SPLINE
SPL {X  -134.737, Y  +296.229, Z    +0.000, E1  +312.110, E3 -135435.927}
SPL {X  -154.917, Y  +342.531, Z    +0.000, E1  +328.797, E3 -135454.495}
SPL {X  -159.440, Y  +369.246, Z    +0.000, E1  +346.542, E3 -135458.394}
SPL {X  -159.987, Y  +381.470, Z    +0.000, E1  +357.024, E3 -135458.993}
SPL {X  -159.990, Y  +384.500, Z    +0.000, E1  +360.000, E3 -135459.026}
SPL {X  -159.990, Y  +386.323, Z    +0.000, E1  +363.079, E3 -135459.048}
SPL {X  -159.990, Y  +390.285, Z    +0.000, E1  +371.315, E3 -135459.169}
SPL {X  -159.990, Y  +394.559, Z    +0.000, E1  +380.770, E3 -135459.431}
SPL {X  -159.990, Y  +399.334, Z    +0.000, E1  +390.876, E3 -135459.870}
SPL {X  -159.990, Y  +405.006, Z    +0.000, E1  +400.810, E3 -135460.588}
SPL {X  -159.990, Y  +415.193, Z    +0.000, E1  +412.724, E3 -135462.475}
SPL {X  -159.990, Y  +465.395, Z    +0.000, E1  +428.959, E3 -135477.563}
SPL {X  -159.990, Y  +657.157, Z    +0.000, E1  +432.499, E3 -135573.960}
SPL {X  -159.693, Y  +681.249, Z    +0.000, E1  +432.488, E3 -135590.354}
SPL {X  -157.599, Y  +699.059, Z    +0.000, E1  +432.249, E3 -135604.514}
SPL {X  -155.217, Y  +710.289, Z    +0.000, E1  +431.989, E3 -135614.530}
SPL {X  -152.611, Y  +719.527, Z    +0.000, E1  +431.702, E3 -135623.352}
SPL {X  -149.536, Y  +728.383, Z    +0.000, E1  +431.359, E3 -135632.331}
SPL {X  -146.250, Y  +736.367, Z    +0.000, E1  +430.965, E3 -135640.885}
SPL {X  -143.481, Y  +742.281, Z    +0.000, E1  +430.623, E3 -135647.480}
SPL {X  -140.071, Y  +748.811, Z    +0.000, E1  +430.193, E3 -135654.992}
SPL {X  -136.578, Y  +754.826, Z    +0.000, E1  +429.723, E3 -135662.122}
SPL {X  -132.176, Y  +761.646, Z    +0.000, E1  +429.128, E3 -135670.365}
SPL {X  -127.941, Y  +767.561, Z    +0.000, E1  +428.475, E3 -135677.673}
SPL {X  -124.983, Y  +771.380, Z    +0.000, E1  +428.003, E3 -135682.392}
SPL {X  -122.624, Y  +774.263, Z    +0.000, E1  +427.622, E3 -135685.915}
SPL {X   -84.435, Y  +807.395, Z    +0.000, E1  +415.948, E3 -135796.919}
ENDSPLINE

SPLINE
SPL {X  -119.703, Y  +777.650, Z    +0.000, E1  +411.831, E3 -135960.926}
SPL {X  -145.184, Y  +738.720, Z    +0.000, E1  +403.488, E3 -135987.484}
SPL {X  -156.175, Y  +706.232, Z    +0.000, E1  +388.819, E3 -135996.369}
SPL {X  -159.337, Y  +685.942, Z    +0.000, E1  +374.672, E3 -135998.920}
SPL {X  -159.962, Y  +674.468, Z    +0.000, E1  +364.846, E3 -135999.539}
SPL {X  -159.990, Y  +669.479, Z    +0.000, E1  +359.996, E3 -135999.613}
SPL {X  -159.990, Y  +667.035, Z    +0.000, E1  +355.461, E3 -135999.644}
SPL {X  -159.990, Y  +662.914, Z    +0.000, E1  +346.506, E3 -135999.782}
SPL {X  -159.990, Y  +658.254, Z    +0.000, E1  +335.847, E3 -136000.060}
SPL {X  -159.990, Y  +650.381, Z    +0.000, E1  +320.607, E3 -136000.912}
SPL {X  -159.990, Y  +638.701, Z    +0.000, E1  +306.047, E3 -136002.798}
SPL {X  -159.990, Y  +618.566, Z    +0.000, E1  +295.881, E3 -136008.306}
SPL {X  -159.990, Y  +582.261, Z    +0.000, E1  +290.657, E3 -136021.792}
SPL {X  -159.990, Y  +406.555, Z    +0.000, E1  +288.365, E3 -136118.038}
SPL {X  -159.990, Y  +385.723, Z    +0.000, E1  +288.390, E3 -136132.777}
SPL {X  -159.404, Y  +368.814, Z    +0.000, E1  +288.444, E3 -136145.306}
SPL {X  -157.440, Y  +354.048, Z    +0.000, E1  +288.658, E3 -136157.779}
SPL {X  -155.889, Y  +346.508, Z    +0.000, E1  +289.539, E3 -136171.327}
SPL {X  -154.332, Y  +340.328, Z    +0.000, E1  +289.976, E3 -136179.555}
SPL {X  -150.579, Y  +328.438, Z    +0.000, E1  +289.626, E3 -136185.274}
SPL {X  -146.933, Y  +319.195, Z    +0.000, E1  +289.770, E3 -136192.965}
SPL {X  -143.573, Y  +311.906, Z    +0.000, E1  +290.194, E3 -136201.275}
SPL {X  -139.693, Y  +304.508, Z    +0.000, E1  +290.699, E3 -136210.003}
SPL {X  -135.622, Y  +297.627, Z    +0.000, E1  +291.269, E3 -136218.411}
SPL {X  -131.165, Y  +290.889, Z    +0.000, E1  +291.906, E3 -136226.797}
SPL {X  -126.457, Y  +284.492, Z    +0.000, E1  +292.648, E3 -136234.882}
SPL {X  -123.432, Y  +280.710, Z    +0.000, E1  +293.170, E3 -136239.668}
SPL {X   -85.607, Y  +247.340, Z    +0.000, E1  +306.083, E3 -136381.389}
ENDSPLINE

SPLINE
SPL {X  -134.737, Y  +296.229, Z    +0.000, E1  +312.110, E3 -136524.162}
SPL {X  -154.917, Y  +342.531, Z    +0.000, E1  +328.797, E3 -136542.730}
SPL {X  -159.440, Y  +369.246, Z    +0.000, E1  +346.542, E3 -136546.629}
SPL {X  -159.987, Y  +381.470, Z    +0.000, E1  +357.024, E3 -136547.228}
SPL {X  -159.990, Y  +384.500, Z    +0.000, E1  +360.000, E3 -136547.261}
SPL {X  -159.990, Y  +386.323, Z    +0.000, E1  +363.079, E3 -136547.283}
SPL {X  -159.990, Y  +390.285, Z    +0.000, E1  +371.315, E3 -136547.404}
SPL {X  -159.990, Y  +394.559, Z    +0.000, E1  +380.770, E3 -136547.666}
SPL {X  -159.990, Y  +402.118, Z    +0.000, E1  +395.793, E3 -136548.457}
SPL {X  -159.990, Y  +415.193, Z    +0.000, E1  +412.724, E3 -136550.710}
SPL {X  -159.990, Y  +465.395, Z    +0.000, E1  +428.959, E3 -136565.799}
SPL {X  -159.990, Y  +652.170, Z    +0.000, E1  +432.485, E3 -136658.894}
SPL {X  -159.990, Y  +670.864, Z    +0.000, E1  +432.509, E3 -136671.342}
SPL {X  -159.251, Y  +686.856, Z    +0.000, E1  +432.412, E3 -136682.884}
SPL {X  -157.599, Y  +699.059, Z    +0.000, E1  +432.249, E3 -136692.749}
SPL {X  -155.217, Y  +710.289, Z    +0.000, E1  +431.989, E3 -136702.766}
SPL {X  -152.611, Y  +719.527, Z    +0.000, E1  +431.702, E3 -136711.587}
SPL {X  -149.536, Y  +728.383, Z    +0.000, E1  +431.359, E3 -136720.566}
SPL {X  -146.250, Y  +736.367, Z    +0.000, E1  +430.965, E3 -136729.120}
SPL {X  -143.481, Y  +742.281, Z    +0.000, E1  +430.623, E3 -136735.716}
SPL {X  -140.071, Y  +748.811, Z    +0.000, E1  +430.193, E3 -136743.227}
SPL {X  -136.578, Y  +754.826, Z    +0.000, E1  +429.723, E3 -136750.357}
SPL {X  -133.265, Y  +760.028, Z    +0.000, E1  +429.258, E3 -136756.658}
SPL {X  -129.890, Y  +764.909, Z    +0.000, E1  +428.775, E3 -136762.628}
SPL {X  -125.802, Y  +770.346, Z    +0.000, E1  +428.156, E3 -136769.328}
SPL {X  -122.624, Y  +774.263, Z    +0.000, E1  +427.622, E3 -136774.150}
SPL {X   -84.435, Y  +807.395, Z    +0.000, E1  +415.948, E3 -136885.155}
ENDSPLINE

SPLINE
SPL {X  -119.703, Y  +777.650, Z    +0.000, E1  +411.831, E3 -137049.161}
SPL {X  -145.184, Y  +738.720, Z    +0.000, E1  +403.488, E3 -137075.719}
SPL {X  -156.175, Y  +706.232, Z    +0.000, E1  +388.819, E3 -137084.604}
SPL {X  -159.337, Y  +685.942, Z    +0.000, E1  +374.672, E3 -137087.155}
SPL {X  -159.962, Y  +674.468, Z    +0.000, E1  +364.846, E3 -137087.774}
SPL {X  -159.990, Y  +669.479, Z    +0.000, E1  +359.996, E3 -137087.848}
SPL {X  -159.990, Y  +667.035, Z    +0.000, E1  +355.461, E3 -137087.879}
SPL {X  -159.990, Y  +662.914, Z    +0.000, E1  +346.506, E3 -137088.018}
SPL {X  -159.990, Y  +658.254, Z    +0.000, E1  +335.847, E3 -137088.295}
SPL {X  -159.990, Y  +652.944, Z    +0.000, E1  +324.878, E3 -137088.799}
SPL {X  -159.990, Y  +642.509, Z    +0.000, E1  +309.910, E3 -137090.371}
SPL {X  -159.990, Y  +618.566, Z    +0.000, E1  +295.881, E3 -137096.541}
SPL {X  -159.990, Y  +584.545, Z    +0.000, E1  +290.812, E3 -137109.076}
SPL {X  -159.990, Y  +578.002, Z    +0.000, E1  +290.393, E3 -137111.800}
SPL {X  -159.990, Y  +426.570, Z    +0.000, E1  +288.401, E3 -137192.290}
SPL {X  -159.990, Y  +405.946, Z    +0.000, E1  +288.370, E3 -137206.720}
SPL {X  -159.967, Y  +379.776, Z    +0.000, E1  +288.366, E3 -137225.167}
SPL {X  -158.535, Y  +360.970, Z    +0.000, E1  +288.540, E3 -137239.989}
SPL {X  -156.277, Y  +348.230, Z    +0.000, E1  +288.789, E3 -137251.332}
SPL {X  -155.351, Y  +344.251, Z    +0.000, E1  +289.996, E3 -137265.124}
SPL {X  -150.579, Y  +328.438, Z    +0.000, E1  +289.626, E3 -137273.509}
SPL {X  -146.933, Y  +319.195, Z    +0.000, E1  +289.770, E3 -137281.200}
SPL {X  -143.573, Y  +311.906, Z    +0.000, E1  +290.194, E3 -137289.510}
SPL {X  -139.693, Y  +304.508, Z    +0.000, E1  +290.699, E3 -137298.239}
SPL {X  -135.622, Y  +297.627, Z    +0.000, E1  +291.269, E3 -137306.647}
SPL {X  -131.165, Y  +290.889, Z    +0.000, E1  +291.906, E3 -137315.032}
SPL {X  -126.457, Y  +284.492, Z    +0.000, E1  +292.648, E3 -137323.118}
SPL {X  -123.432, Y  +280.710, Z    +0.000, E1  +293.170, E3 -137327.903}
SPL {X   -85.607, Y  +247.340, Z    +0.000, E1  +306.083, E3 -137469.625}
ENDSPLINE

SPLINE
SPL {X  -134.737, Y  +296.229, Z    +0.000, E1  +312.110, E3 -137612.398}
SPL {X  -154.917, Y  +342.531, Z    +0.000, E1  +328.797, E3 -137630.965}
SPL {X  -159.440, Y  +369.246, Z    +0.000, E1  +346.542, E3 -137634.864}
SPL {X  -159.957, Y  +379.264, Z    +0.000, E1  +355.091, E3 -137635.421}
SPL {X  -159.990, Y  +384.670, Z    +0.000, E1  +360.079, E3 -137635.498}
SPL {X  -159.990, Y  +389.248, Z    +0.000, E1  +368.879, E3 -137635.602}
SPL {X  -159.990, Y  +394.559, Z    +0.000, E1  +380.770, E3 -137635.901}
SPL {X  -159.990, Y  +402.118, Z    +0.000, E1  +395.793, E3 -137636.693}
SPL {X  -159.990, Y  +415.193, Z    +0.000, E1  +412.724, E3 -137638.945}
SPL {X  -159.990, Y  +465.395, Z    +0.000, E1  +428.959, E3 -137654.034}
SPL {X  -159.990, Y  +657.157, Z    +0.000, E1  +432.499, E3 -137750.431}
SPL {X  -159.947, Y  +675.227, Z    +0.000, E1  +432.487, E3 -137762.591}
SPL {X  -159.251, Y  +686.856, Z    +0.000, E1  +432.412, E3 -137771.119}
SPL {X  -157.599, Y  +699.059, Z    +0.000, E1  +432.249, E3 -137780.984}
SPL {X  -155.217, Y  +710.289, Z    +0.000, E1  +431.989, E3 -137791.001}
SPL {X  -152.611, Y  +719.527, Z    +0.000, E1  +431.702, E3 -137799.822}
SPL {X  -149.536, Y  +728.383, Z    +0.000, E1  +431.359, E3 -137808.801}
SPL {X  -146.250, Y  +736.367, Z    +0.000, E1  +430.965, E3 -137817.356}
SPL {X  -143.481, Y  +742.281, Z    +0.000, E1  +430.623, E3 -137823.951}
SPL {X  -140.071, Y  +748.811, Z    +0.000, E1  +430.193, E3 -137831.463}
SPL {X  -136.578, Y  +754.826, Z    +0.000, E1  +429.723, E3 -137838.592}
SPL {X  -133.265, Y  +760.028, Z    +0.000, E1  +429.258, E3 -137844.893}
SPL {X  -129.890, Y  +764.909, Z    +0.000, E1  +428.775, E3 -137850.864}
SPL {X  -125.802, Y  +770.346, Z    +0.000, E1  +428.156, E3 -137857.563}
SPL {X  -122.624, Y  +774.263, Z    +0.000, E1  +427.622, E3 -137862.386}
SPL {X   -84.435, Y  +807.395, Z    +0.000, E1  +415.948, E3 -137973.390}
ENDSPLINE

SPLINE
SPL {X  -119.703, Y  +777.650, Z    +0.000, E1  +411.831, E3 -138137.397}
SPL {X  -145.184, Y  +738.720, Z    +0.000, E1  +403.488, E3 -138163.955}
SPL {X  -154.467, Y  +713.173, Z    +0.000, E1  +392.658, E3 -138171.550}
SPL {X  -157.530, Y  +699.446, Z    +0.000, E1  +384.482, E3 -138173.966}
SPL {X  -159.337, Y  +685.942, Z    +0.000, E1  +374.672, E3 -138175.391}
SPL {X  -159.962, Y  +674.468, Z    +0.000, E1  +364.846, E3 -138176.009}
SPL {X  -159.990, Y  +669.479, Z    +0.000, E1  +359.996, E3 -138176.083}
SPL {X  -159.990, Y  +667.035, Z    +0.000, E1  +355.461, E3 -138176.114}
SPL {X  -159.990, Y  +662.914, Z    +0.000, E1  +346.506, E3 -138176.253}
SPL {X  -159.990, Y  +658.254, Z    +0.000, E1  +335.847, E3 -138176.531}
SPL {X  -159.990, Y  +652.944, Z    +0.000, E1  +324.878, E3 -138177.034}
SPL {X  -159.990, Y  +642.509, Z    +0.000, E1  +309.910, E3 -138178.606}
SPL {X  -159.990, Y  +618.566, Z    +0.000, E1  +295.881, E3 -138184.777}
SPL {X  -159.990, Y  +582.261, Z    +0.000, E1  +290.657, E3 -138198.262}
SPL {X  -159.990, Y  +406.555, Z    +0.000, E1  +288.365, E3 -138294.509}
SPL {X  -159.990, Y  +385.723, Z    +0.000, E1  +288.390, E3 -138309.247}
SPL {X  -159.700, Y  +372.863, Z    +0.000, E1  +288.430, E3 -138318.653}
SPL {X  -158.535, Y  +360.970, Z    +0.000, E1  +288.540, E3 -138328.224}
SPL {X  -156.277, Y  +348.230, Z    +0.000, E1  +288.789, E3 -138339.567}
SPL {X  -155.351, Y  +344.251, Z    +0.000, E1  +289.996, E3 -138353.359}
SPL {X  -150.579, Y  +328.438, Z    +0.000, E1  +289.626, E3 -138361.744}
SPL {X  -146.933, Y  +319.195, Z    +0.000, E1  +289.770, E3 -138369.435}
SPL {X  -143.573, Y  +311.906, Z    +0.000, E1  +290.194, E3 -138377.746}
SPL {X  -140.547, Y  +306.057, Z    +0.000, E1  +290.601, E3 -138384.638}
SPL {X  -137.438, Y  +300.600, Z    +0.000, E1  +291.016, E3 -138391.232}
SPL {X  -133.397, Y  +294.172, Z    +0.000, E1  +291.584, E3 -138399.167}
SPL {X  -128.822, Y  +287.623, Z    +0.000, E1  +292.271, E3 -138407.391}
SPL {X  -124.502, Y  +282.021, Z    +0.000, E1  +292.965, E3 -138414.465}
SPL {X   -85.607, Y  +247.340, Z    +0.000, E1  +306.083, E3 -138557.860}
ENDSPLINE

SPLINE
SPL {X  -119.557, Y  +276.184, Z    +0.000, E1  +308.968, E3 -138681.397}
SPL {X  -138.294, Y  +302.054, Z    +0.000, E1  +313.424, E3 -138704.719}
SPL {X  -153.211, Y  +336.421, Z    +0.000, E1  +325.738, E3 -138717.841}
SPL {X  -158.240, Y  +358.900, Z    +0.000, E1  +338.911, E3 -138722.046}
SPL {X  -159.674, Y  +372.451, Z    +0.000, E1  +349.222, E3 -138723.342}
SPL {X  -159.987, Y  +381.470, Z    +0.000, E1  +357.024, E3 -138723.699}
SPL {X  -159.990, Y  +384.761, Z    +0.000, E1  +360.257, E3 -138723.734}
SPL {X  -159.990, Y  +389.248, Z    +0.000, E1  +368.879, E3 -138723.838}
SPL {X  -159.990, Y  +394.559, Z    +0.000, E1  +380.770, E3 -138724.137}
SPL {X  -159.990, Y  +402.118, Z    +0.000, E1  +395.793, E3 -138724.928}
SPL {X  -159.990, Y  +415.193, Z    +0.000, E1  +412.724, E3 -138727.181}
SPL {X  -159.990, Y  +465.395, Z    +0.000, E1  +428.959, E3 -138742.269}
SPL {X  -159.990, Y  +657.157, Z    +0.000, E1  +432.499, E3 -138838.666}
SPL {X  -159.693, Y  +681.249, Z    +0.000, E1  +432.488, E3 -138855.060}
SPL {X  -157.599, Y  +699.059, Z    +0.000, E1  +432.249, E3 -138869.220}
SPL {X  -155.217, Y  +710.289, Z    +0.000, E1  +431.989, E3 -138879.236}
SPL {X  -152.611, Y  +719.527, Z    +0.000, E1  +431.702, E3 -138888.058}
SPL {X  -149.536, Y  +728.383, Z    +0.000, E1  +431.359, E3 -138897.037}
SPL {X  -146.250, Y  +736.367, Z    +0.000, E1  +430.965, E3 -138905.591}
SPL {X  -143.481, Y  +742.281, Z    +0.000, E1  +430.623, E3 -138912.186}
SPL {X  -140.071, Y  +748.811, Z    +0.000, E1  +430.193, E3 -138919.698}
SPL {X  -136.578, Y  +754.826, Z    +0.000, E1  +429.723, E3 -138926.827}
SPL {X  -133.265, Y  +760.028, Z    +0.000, E1  +429.258, E3 -138933.128}
SPL {X  -129.890, Y  +764.909, Z    +0.000, E1  +428.775, E3 -138939.099}
SPL {X  -125.802, Y  +770.346, Z    +0.000, E1  +428.156, E3 -138945.798}
SPL {X  -122.624, Y  +774.263, Z    +0.000, E1  +427.622, E3 -138950.621}
SPL {X   -84.435, Y  +807.395, Z    +0.000, E1  +415.948, E3 -139061.625}
ENDSPLINE

SPLINE
SPL {X  -119.703, Y  +777.650, Z    +0.000, E1  +411.831, E3 -139225.632}
SPL {X  -145.184, Y  +738.720, Z    +0.000, E1  +403.488, E3 -139252.190}
SPL {X  -156.175, Y  +706.232, Z    +0.000, E1  +388.819, E3 -139261.075}
SPL {X  -159.337, Y  +685.942, Z    +0.000, E1  +374.672, E3 -139263.626}
SPL {X  -159.900, Y  +676.871, Z    +0.000, E1  +366.955, E3 -139264.174}
SPL {X  -159.990, Y  +669.634, Z    +0.000, E1  +360.285, E3 -139264.318}
SPL {X  -159.990, Y  +667.035, Z    +0.000, E1  +355.461, E3 -139264.349}
SPL {X  -159.990, Y  +662.914, Z    +0.000, E1  +346.506, E3 -139264.488}
SPL {X  -159.990, Y  +658.254, Z    +0.000, E1  +335.847, E3 -139264.766}
SPL {X  -159.990, Y  +652.944, Z    +0.000, E1  +324.878, E3 -139265.270}
SPL {X  -159.990, Y  +642.509, Z    +0.000, E1  +309.910, E3 -139266.841}
SPL {X  -159.990, Y  +618.566, Z    +0.000, E1  +295.881, E3 -139273.012}
SPL {X  -159.990, Y  +584.545, Z    +0.000, E1  +290.812, E3 -139285.547}
SPL {X  -159.990, Y  +578.002, Z    +0.000, E1  +290.393, E3 -139288.271}
SPL {X  -159.990, Y  +426.570, Z    +0.000, E1  +288.401, E3 -139368.761}
SPL {X  -159.990, Y  +405.946, Z    +0.000, E1  +288.370, E3 -139383.191}
SPL {X  -159.967, Y  +379.776, Z    +0.000, E1  +288.366, E3 -139401.637}
SPL {X  -158.535, Y  +360.970, Z    +0.000, E1  +288.540, E3 -139416.459}
SPL {X  -156.882, Y  +351.118, Z    +0.000, E1  +288.737, E3 -139425.171}
SPL {X  -155.538, Y  +345.018, Z    +0.000, E1  +288.891, E3 -139430.878}
SPL {X  -155.351, Y  +344.251, Z    +0.000, E1  +289.996, E3 -139441.594}
SPL {X  -150.579, Y  +328.438, Z    +0.000, E1  +289.626, E3 -139449.980}
SPL {X  -146.933, Y  +319.195, Z    +0.000, E1  +289.770, E3 -139457.671}
SPL {X  -143.573, Y  +311.906, Z    +0.000, E1  +290.194, E3 -139465.981}
SPL {X  -140.547, Y  +306.057, Z    +0.000, E1  +290.601, E3 -139472.873}
SPL {X  -137.438, Y  +300.600, Z    +0.000, E1  +291.016, E3 -139479.467}
SPL {X  -133.397, Y  +294.172, Z    +0.000, E1  +291.584, E3 -139487.402}
SPL {X  -128.822, Y  +287.623, Z    +0.000, E1  +292.271, E3 -139495.627}
SPL {X  -124.502, Y  +282.021, Z    +0.000, E1  +292.965, E3 -139502.701}
SPL {X   -85.607, Y  +247.340, Z    +0.000, E1  +306.083, E3 -139646.095}
ENDSPLINE

SPLINE
SPL {X  -134.737, Y  +296.229, Z    +0.000, E1  +312.110, E3 -139788.868}
SPL {X  -153.211, Y  +336.421, Z    +0.000, E1  +325.738, E3 -139806.076}
SPL {X  -158.240, Y  +358.900, Z    +0.000, E1  +338.911, E3 -139810.281}
SPL {X  -159.854, Y  +375.896, Z    +0.000, E1  +352.019, E3 -139811.747}
SPL {X  -159.990, Y  +384.398, Z    +0.000, E1  +359.828, E3 -139811.967}
SPL {X  -159.990, Y  +386.323, Z    +0.000, E1  +363.079, E3 -139811.989}
SPL {X  -159.990, Y  +390.285, Z    +0.000, E1  +371.315, E3 -139812.110}
SPL {X  -159.990, Y  +394.559, Z    +0.000, E1  +380.770, E3 -139812.372}
SPL {X  -159.990, Y  +399.334, Z    +0.000, E1  +390.876, E3 -139812.811}
SPL {X  -159.990, Y  +405.006, Z    +0.000, E1  +400.810, E3 -139813.529}
SPL {X  -159.990, Y  +415.193, Z    +0.000, E1  +412.724, E3 -139815.416}
SPL {X  -159.990, Y  +465.395, Z    +0.000, E1  +428.959, E3 -139830.505}
SPL {X  -159.990, Y  +657.157, Z    +0.000, E1  +432.499, E3 -139926.901}
SPL {X  -159.693, Y  +681.249, Z    +0.000, E1  +432.488, E3 -139943.295}
SPL {X  -157.599, Y  +699.059, Z    +0.000, E1  +432.249, E3 -139957.455}
SPL {X  -155.217, Y  +710.289, Z    +0.000, E1  +431.989, E3 -139967.472}
SPL {X  -152.611, Y  +719.527, Z    +0.000, E1  +431.702, E3 -139976.293}
SPL {X  -149.536, Y  +728.383, Z    +0.000, E1  +431.359, E3 -139985.272}
SPL {X  -146.250, Y  +736.367, Z    +0.000, E1  +430.965, E3 -139993.826}
SPL {X  -143.481, Y  +742.281, Z    +0.000, E1  +430.623, E3 -140000.422}
SPL {X  -140.071, Y  +748.811, Z    +0.000, E1  +430.193, E3 -140007.933}
SPL {X  -136.578, Y  +754.826, Z    +0.000, E1  +429.723, E3 -140015.063}
SPL {X  -133.265, Y  +760.028, Z    +0.000, E1  +429.258, E3 -140021.364}
SPL {X  -129.890, Y  +764.909, Z    +0.000, E1  +428.775, E3 -140027.334}
SPL {X  -125.802, Y  +770.346, Z    +0.000, E1  +428.156, E3 -140034.033}
SPL {X  -122.624, Y  +774.263, Z    +0.000, E1  +427.622, E3 -140038.856}
SPL {X   -84.435, Y  +807.395, Z    +0.000, E1  +415.948, E3 -140149.861}
ENDSPLINE

SPLINE
SPL {X  -119.703, Y  +777.650, Z    +0.000, E1  +411.831, E3 -140313.867}
SPL {X  -145.184, Y  +738.720, Z    +0.000, E1  +403.488, E3 -140340.425}
SPL {X  -156.175, Y  +706.232, Z    +0.000, E1  +388.819, E3 -140349.310}
SPL {X  -159.337, Y  +685.942, Z    +0.000, E1  +374.672, E3 -140351.861}
SPL {X  -159.900, Y  +676.871, Z    +0.000, E1  +366.955, E3 -140352.409}
SPL {X  -159.990, Y  +669.634, Z    +0.000, E1  +360.285, E3 -140352.553}
SPL {X  -159.990, Y  +667.035, Z    +0.000, E1  +355.461, E3 -140352.585}
SPL {X  -159.990, Y  +662.914, Z    +0.000, E1  +346.506, E3 -140352.724}
SPL {X  -159.990, Y  +658.254, Z    +0.000, E1  +335.847, E3 -140353.001}
SPL {X  -159.990, Y  +652.944, Z    +0.000, E1  +324.878, E3 -140353.505}
SPL {X  -159.990, Y  +646.557, Z    +0.000, E1  +314.610, E3 -140354.372}
SPL {X  -159.990, Y  +638.701, Z    +0.000, E1  +306.047, E3 -140355.739}
SPL {X  -159.990, Y  +618.566, Z    +0.000, E1  +295.881, E3 -140361.247}
SPL {X  -159.990, Y  +582.261, Z    +0.000, E1  +290.657, E3 -140374.733}
SPL {X  -159.990, Y  +414.423, Z    +0.000, E1  +288.398, E3 -140465.516}
SPL {X  -159.990, Y  +400.357, Z    +0.000, E1  +288.396, E3 -140475.427}
SPL {X  -159.990, Y  +385.723, Z    +0.000, E1  +288.390, E3 -140485.718}
SPL {X  -159.404, Y  +368.814, Z    +0.000, E1  +288.444, E3 -140498.247}
SPL {X  -157.440, Y  +354.048, Z    +0.000, E1  +288.658, E3 -140510.720}
SPL {X  -155.889, Y  +346.508, Z    +0.000, E1  +289.539, E3 -140524.268}
SPL {X  -154.332, Y  +340.328, Z    +0.000, E1  +289.976, E3 -140532.496}
SPL {X  -150.579, Y  +328.438, Z    +0.000, E1  +289.626, E3 -140538.215}
SPL {X  -146.933, Y  +319.195, Z    +0.000, E1  +289.770, E3 -140545.906}
SPL {X  -143.573, Y  +311.906, Z    +0.000, E1  +290.194, E3 -140554.216}
SPL {X  -139.693, Y  +304.508, Z    +0.000, E1  +290.699, E3 -140562.945}
SPL {X  -135.622, Y  +297.627, Z    +0.000, E1  +291.269, E3 -140571.353}
SPL {X  -132.531, Y  +292.877, Z    +0.000, E1  +291.734, E3 -140577.288}
SPL {X  -128.822, Y  +287.623, Z    +0.000, E1  +292.271, E3 -140583.862}
SPL {X  -124.502, Y  +282.021, Z    +0.000, E1  +292.965, E3 -140590.936}
SPL {X   -85.607, Y  +247.340, Z    +0.000, E1  +306.083, E3 -140734.331}
ENDSPLINE

SPLINE
SPL {X  -134.737, Y  +296.229, Z    +0.000, E1  +312.110, E3 -140877.103}
SPL {X  -154.917, Y  +342.531, Z    +0.000, E1  +328.797, E3 -140895.671}
SPL {X  -159.440, Y  +369.246, Z    +0.000, E1  +346.542, E3 -140899.570}
SPL {X  -159.987, Y  +381.470, Z    +0.000, E1  +357.024, E3 -140900.169}
SPL {X  -159.990, Y  +384.500, Z    +0.000, E1  +360.000, E3 -140900.203}
SPL {X  -159.990, Y  +386.323, Z    +0.000, E1  +363.079, E3 -140900.224}
SPL {X  -159.990, Y  +390.285, Z    +0.000, E1  +371.315, E3 -140900.345}
SPL {X  -159.990, Y  +394.559, Z    +0.000, E1  +380.770, E3 -140900.607}
SPL {X  -159.990, Y  +402.118, Z    +0.000, E1  +395.793, E3 -140901.399}
SPL {X  -159.990, Y  +415.193, Z    +0.000, E1  +412.724, E3 -140903.651}
SPL {X  -159.990, Y  +465.395, Z    +0.000, E1  +428.959, E3 -140918.740}
SPL {X  -159.990, Y  +657.157, Z    +0.000, E1  +432.499, E3 -141015.137}
SPL {X  -159.693, Y  +681.249, Z    +0.000, E1  +432.488, E3 -141031.531}
SPL {X  -157.599, Y  +699.059, Z    +0.000, E1  +432.249, E3 -141045.690}
SPL {X  -155.217, Y  +710.289, Z    +0.000, E1  +431.989, E3 -141055.707}
SPL {X  -152.611, Y  +719.527, Z    +0.000, E1  +431.702, E3 -141064.528}
SPL {X  -149.536, Y  +728.383, Z    +0.000, E1  +431.359, E3 -141073.507}
SPL {X  -146.250, Y  +736.367, Z    +0.000, E1  +430.965, E3 -141082.061}
SPL {X  -143.481, Y  +742.281, Z    +0.000, E1  +430.623, E3 -141088.657}
SPL {X  -140.071, Y  +748.811, Z    +0.000, E1  +430.193, E3 -141096.169}
SPL {X  -136.578, Y  +754.826, Z    +0.000, E1  +429.723, E3 -141103.298}
SPL {X  -133.265, Y  +760.028, Z    +0.000, E1  +429.258, E3 -141109.599}
SPL {X  -129.890, Y  +764.909, Z    +0.000, E1  +428.775, E3 -141115.570}
SPL {X  -125.802, Y  +770.346, Z    +0.000, E1  +428.156, E3 -141122.269}
SPL {X  -122.624, Y  +774.263, Z    +0.000, E1  +427.622, E3 -141127.091}
SPL {X   -84.435, Y  +807.395, Z    +0.000, E1  +415.948, E3 -141238.096}
ENDSPLINE

SPLINE
SPL {X  -119.703, Y  +777.650, Z    +0.000, E1  +411.831, E3 -141402.103}
SPL {X  -145.184, Y  +738.720, Z    +0.000, E1  +403.488, E3 -141428.661}
SPL {X  -156.175, Y  +706.232, Z    +0.000, E1  +388.819, E3 -141437.545}
SPL {X  -159.337, Y  +685.942, Z    +0.000, E1  +374.672, E3 -141440.097}
SPL {X  -159.962, Y  +674.468, Z    +0.000, E1  +364.846, E3 -141440.715}
SPL {X  -159.990, Y  +669.479, Z    +0.000, E1  +359.996, E3 -141440.789}
SPL {X  -159.990, Y  +667.035, Z    +0.000, E1  +355.461, E3 -141440.820}
SPL {X  -159.990, Y  +662.914, Z    +0.000, E1  +346.506, E3 -141440.959}
SPL {X  -159.990, Y  +658.254, Z    +0.000, E1  +335.847, E3 -141441.237}
SPL {X  -159.990, Y  +652.944, Z    +0.000, E1  +324.878, E3 -141441.740}
SPL {X  -159.990, Y  +642.509, Z    +0.000, E1  +309.910, E3 -141443.312}
SPL {X  -159.990, Y  +618.566, Z    +0.000, E1  +295.881, E3 -141449.482}
SPL {X  -159.990, Y  +584.545, Z    +0.000, E1  +290.812, E3 -141462.018}
SPL {X  -159.990, Y  +578.002, Z    +0.000, E1  +290.393, E3 -141464.741}
SPL {X  -159.990, Y  +426.570, Z    +0.000, E1  +288.401, E3 -141545.231}
SPL {X  -159.990, Y  +405.946, Z    +0.000, E1  +288.370, E3 -141559.661}
SPL {X  -159.967, Y  +379.776, Z    +0.000, E1  +288.366, E3 -141578.108}
SPL {X  -158.535, Y  +360.970, Z    +0.000, E1  +288.540, E3 -141592.930}
SPL {X  -156.277, Y  +348.230, Z    +0.000, E1  +288.789, E3 -141604.273}
SPL {X  -155.351, Y  +344.251, Z    +0.000, E1  +289.996, E3 -141618.065}
SPL {X  -150.579, Y  +328.438, Z    +0.000, E1  +289.626, E3 -141626.450}
SPL {X  -146.933, Y  +319.195, Z    +0.000, E1  +289.770, E3 -141634.141}
SPL {X  -143.573, Y  +311.906, Z    +0.000, E1  +290.194, E3 -141642.452}
SPL {X  -139.693, Y  +304.508, Z    +0.000, E1  +290.699, E3 -141651.180}
SPL {X  -135.622, Y  +297.627, Z    +0.000, E1  +291.269, E3 -141659.588}
SPL {X  -131.165, Y  +290.889, Z    +0.000, E1  +291.906, E3 -141667.973}
SPL {X  -126.457, Y  +284.492, Z    +0.000, E1  +292.648, E3 -141676.059}
SPL {X  -123.432, Y  +280.710, Z    +0.000, E1  +293.170, E3 -141680.845}
SPL {X   -85.607, Y  +247.340, Z    +0.000, E1  +306.083, E3 -141822.566}
ENDSPLINE

SPLINE
SPL {X  -134.737, Y  +296.229, Z    +0.000, E1  +312.110, E3 -141965.339}
SPL {X  -154.917, Y  +342.531, Z    +0.000, E1  +328.797, E3 -141983.906}
SPL {X  -159.440, Y  +369.246, Z    +0.000, E1  +346.542, E3 -141987.806}
SPL {X  -159.987, Y  +381.470, Z    +0.000, E1  +357.024, E3 -141988.405}
SPL {X  -159.990, Y  +384.500, Z    +0.000, E1  +360.000, E3 -141988.438}
SPL {X  -159.990, Y  +386.323, Z    +0.000, E1  +363.079, E3 -141988.459}
SPL {X  -159.990, Y  +390.285, Z    +0.000, E1  +371.315, E3 -141988.580}
SPL {X  -159.990, Y  +394.559, Z    +0.000, E1  +380.770, E3 -141988.843}
SPL {X  -159.990, Y  +402.118, Z    +0.000, E1  +395.793, E3 -141989.634}
SPL {X  -159.990, Y  +415.193, Z    +0.000, E1  +412.724, E3 -141991.886}
SPL {X  -159.990, Y  +465.395, Z    +0.000, E1  +428.959, E3 -142006.975}
SPL {X  -159.990, Y  +657.157, Z    +0.000, E1  +432.499, E3 -142103.372}
SPL {X  -159.693, Y  +681.249, Z    +0.000, E1  +432.488, E3 -142119.766}
SPL {X  -157.599, Y  +699.059, Z    +0.000, E1  +432.249, E3 -142133.926}
SPL {X  -155.217, Y  +710.289, Z    +0.000, E1  +431.989, E3 -142143.942}
SPL {X  -152.611, Y  +719.527, Z    +0.000, E1  +431.702, E3 -142152.763}
SPL {X  -149.536, Y  +728.383, Z    +0.000, E1  +431.359, E3 -142161.743}
SPL {X  -146.250, Y  +736.367, Z    +0.000, E1  +430.965, E3 -142170.297}
SPL {X  -143.481, Y  +742.281, Z    +0.000, E1  +430.623, E3 -142176.892}
SPL {X  -140.071, Y  +748.811, Z    +0.000, E1  +430.193, E3 -142184.404}
SPL {X  -136.578, Y  +754.826, Z    +0.000, E1  +429.723, E3 -142191.533}
SPL {X  -133.265, Y  +760.028, Z    +0.000, E1  +429.258, E3 -142197.834}
SPL {X  -129.890, Y  +764.909, Z    +0.000, E1  +428.775, E3 -142203.805}
SPL {X  -125.802, Y  +770.346, Z    +0.000, E1  +428.156, E3 -142210.504}
SPL {X  -122.624, Y  +774.263, Z    +0.000, E1  +427.622, E3 -142215.327}
SPL {X   -84.435, Y  +807.395, Z    +0.000, E1  +415.948, E3 -142326.331}
ENDSPLINE

SPLINE
SPL {X  -119.703, Y  +777.650, Z    +0.000, E1  +411.831, E3 -142490.338}
SPL {X  -145.184, Y  +738.720, Z    +0.000, E1  +403.488, E3 -142516.896}
SPL {X  -156.175, Y  +706.232, Z    +0.000, E1  +388.819, E3 -142525.781}
SPL {X  -159.337, Y  +685.942, Z    +0.000, E1  +374.672, E3 -142528.332}
SPL {X  -159.962, Y  +674.468, Z    +0.000, E1  +364.846, E3 -142528.950}
SPL {X  -159.990, Y  +669.479, Z    +0.000, E1  +359.996, E3 -142529.025}
SPL {X  -159.990, Y  +667.035, Z    +0.000, E1  +355.461, E3 -142529.055}
SPL {X  -159.990, Y  +662.914, Z    +0.000, E1  +346.506, E3 -142529.194}
SPL {X  -159.990, Y  +658.254, Z    +0.000, E1  +335.847, E3 -142529.472}
SPL {X  -159.990, Y  +652.944, Z    +0.000, E1  +324.878, E3 -142529.976}
SPL {X  -159.990, Y  +642.509, Z    +0.000, E1  +309.910, E3 -142531.547}
SPL {X  -159.990, Y  +618.566, Z    +0.000, E1  +295.881, E3 -142537.718}
SPL {X  -159.990, Y  +584.545, Z    +0.000, E1  +290.812, E3 -142550.253}
SPL {X  -159.990, Y  +578.002, Z    +0.000, E1  +290.393, E3 -142552.977}
SPL {X  -159.990, Y  +426.570, Z    +0.000, E1  +288.401, E3 -142633.467}
SPL {X  -159.990, Y  +405.946, Z    +0.000, E1  +288.370, E3 -142647.897}
SPL {X  -159.967, Y  +379.776, Z    +0.000, E1  +288.366, E3 -142666.343}
SPL {X  -158.535, Y  +360.970, Z    +0.000, E1  +288.540, E3 -142681.165}
SPL {X  -156.277, Y  +348.230, Z    +0.000, E1  +288.789, E3 -142692.508}
SPL {X  -155.351, Y  +344.251, Z    +0.000, E1  +289.996, E3 -142706.300}
SPL {X  -150.579, Y  +328.438, Z    +0.000, E1  +289.626, E3 -142714.686}
ENDSPLINE

SPLINE
SPL {X  -153.635, Y  +337.858, Z    +0.000, E1  +292.753, E3 -142732.535}
ENDSPLINE

SPLINE
SPL {X  -150.407, Y  +327.960, Z    +0.000, E1  +293.203, E3 -142744.277}
SPL {X  -146.798, Y  +318.884, Z    +0.000, E1  +293.699, E3 -142755.561}
SPL {X  -142.741, Y  +310.238, Z    +0.000, E1  +294.301, E3 -142766.820}
SPL {X  -139.838, Y  +304.768, Z    +0.000, E1  +294.773, E3 -142774.203}
SPL {X  -137.162, Y  +300.138, Z    +0.000, E1  +295.180, E3 -142780.509}
SPL {X  -132.996, Y  +293.568, Z    +0.000, E1  +295.842, E3 -142789.643}
SPL {X  -128.628, Y  +287.360, Z    +0.000, E1  +296.617, E3 -142798.444}
SPL {X   -98.696, Y  +256.580, Z    +0.000, E1  +308.006, E3 -142935.562}
ENDSPLINE

SPLINE
SPL {X  -138.661, Y  +302.689, Z    +0.000, E1  +316.811, E3 -143053.291}
SPL {X  -154.202, Y  +339.857, Z    +0.000, E1  +330.366, E3 -143070.944}
SPL {X  -158.556, Y  +361.128, Z    +0.000, E1  +342.470, E3 -143075.466}
SPL {X  -159.663, Y  +372.278, Z    +0.000, E1  +350.186, E3 -143076.747}
SPL {X  -159.986, Y  +381.388, Z    +0.000, E1  +357.201, E3 -143077.218}
SPL {X  -159.990, Y  +384.492, Z    +0.000, E1  +359.986, E3 -143077.269}
SPL {X  -159.990, Y  +385.649, Z    +0.000, E1  +361.559, E3 -143077.280}
SPL {X  -159.990, Y  +389.563, Z    +0.000, E1  +367.931, E3 -143077.412}
SPL {X  -159.990, Y  +396.421, Z    +0.000, E1  +380.831, E3 -143077.957}
SPL {X  -159.990, Y  +405.629, Z    +0.000, E1  +396.596, E3 -143079.312}
SPL {X  -159.990, Y  +418.631, Z    +0.000, E1  +410.627, E3 -143082.259}
SPL {X  -159.990, Y  +468.459, Z    +0.000, E1  +425.348, E3 -143101.803}
SPL {X  -159.990, Y  +601.948, Z    +0.000, E1  +428.261, E3 -143187.929}
SPL {X  -159.990, Y  +619.726, Z    +0.000, E1  +428.262, E3 -143202.989}
SPL {X  -159.990, Y  +636.530, Z    +0.000, E1  +428.257, E3 -143217.225}
SPL {X  -159.990, Y  +648.825, Z    +0.000, E1  +428.237, E3 -143227.684}
SPL {X  -159.990, Y  +661.441, Z    +0.000, E1  +428.256, E3 -143238.332}
SPL {X  -159.958, Y  +674.683, Z    +0.000, E1  +428.238, E3 -143249.595}
SPL {X  -159.269, Y  +686.675, Z    +0.000, E1  +428.163, E3 -143260.472}
SPL {X  -157.606, Y  +699.018, Z    +0.000, E1  +427.957, E3 -143272.656}
SPL {X  -155.210, Y  +710.317, Z    +0.000, E1  +427.656, E3 -143284.696}
SPL {X  -152.048, Y  +721.282, Z    +0.000, E1  +427.243, E3 -143297.189}
SPL {X  -148.485, Y  +731.073, Z    +0.000, E1  +426.748, E3 -143309.038}
SPL {X  -145.075, Y  +738.953, Z    +0.000, E1  +426.252, E3 -143319.029}
SPL {X  -141.751, Y  +745.686, Z    +0.000, E1  +425.756, E3 -143327.860}
SPL {X  -138.928, Y  +750.847, Z    +0.000, E1  +425.305, E3 -143334.830}
SPL {X  -136.328, Y  +755.234, Z    +0.000, E1  +424.898, E3 -143340.820}
SPL {X  -132.717, Y  +760.848, Z    +0.000, E1  +424.322, E3 -143348.593}
SPL {X  -128.512, Y  +766.796, Z    +0.000, E1  +423.597, E3 -143356.948}
SPL {X   -99.023, Y  +797.163, Z    +0.000, E1  +413.965, E3 -143458.777}
ENDSPLINE

SPLINE
SPL {X  -130.021, Y  +764.727, Z    +0.000, E1  +405.990, E3 -143598.297}
SPL {X  -148.409, Y  +731.264, Z    +0.000, E1  +396.685, E3 -143622.010}
SPL {X  -155.017, Y  +711.078, Z    +0.000, E1  +387.846, E3 -143629.071}
SPL {X  -158.217, Y  +695.254, Z    +0.000, E1  +378.896, E3 -143632.514}
SPL {X  -159.762, Y  +680.037, Z    +0.000, E1  +368.585, E3 -143634.231}
SPL {X  -159.990, Y  +671.255, Z    +0.000, E1  +361.602, E3 -143634.637}
SPL {X  -159.990, Y  +669.426, Z    +0.000, E1  +359.932, E3 -143634.656}
SPL {X  -159.990, Y  +666.879, Z    +0.000, E1  +356.292, E3 -143634.704}
SPL {X  -159.990, Y  +662.620, Z    +0.000, E1  +348.758, E3 -143634.905}
SPL {X  -159.990, Y  +657.714, Z    +0.000, E1  +339.502, E3 -143635.327}
SPL {X  -159.990, Y  +651.038, Z    +0.000, E1  +327.797, E3 -143636.229}
SPL {X  -159.990, Y  +637.243, Z    +0.000, E1  +311.500, E3 -143639.354}
SPL {X  -159.990, Y  +579.875, Z    +0.000, E1  +294.421, E3 -143662.213}
SPL {X  -159.990, Y  +453.091, Z    +0.000, E1  +291.862, E3 -143745.182}
SPL {X  -159.990, Y  +434.933, Z    +0.000, E1  +291.864, E3 -143760.676}
SPL {X  -159.990, Y  +420.071, Z    +0.000, E1  +291.886, E3 -143773.402}
SPL {X  -159.990, Y  +408.047, Z    +0.000, E1  +291.885, E3 -143783.650}
SPL {X  -159.990, Y  +395.904, Z    +0.000, E1  +291.881, E3 -143793.986}
SPL {X  -157.896, Y  +356.699, Z    +0.000, E1  +289.725, E3 -143806.295}
SPL {X  -156.475, Y  +349.148, Z    +0.000, E1  +290.612, E3 -143819.759}
SPL {X  -155.960, Y  +346.816, Z    +0.000, E1  +291.495, E3 -143828.920}
SPL {X  -154.913, Y  +342.515, Z    +0.000, E1  +292.501, E3 -143840.934}
SPL {X  -152.032, Y  +332.668, Z    +0.000, E1  +292.988, E3 -143852.926}
SPL {X  -148.460, Y  +322.864, Z    +0.000, E1  +293.452, E3 -143864.808}
SPL {X  -144.472, Y  +313.764, Z    +0.000, E1  +294.050, E3 -143876.472}
SPL {X  -140.755, Y  +306.442, Z    +0.000, E1  +294.606, E3 -143886.186}
SPL {X  -137.162, Y  +300.138, Z    +0.000, E1  +295.180, E3 -143894.795}
SPL {X  -134.303, Y  +295.555, Z    +0.000, E1  +295.659, E3 -143901.175}
SPL {X  -131.069, Y  +290.753, Z    +0.000, E1  +296.178, E3 -143907.909}
SPL {X  -127.815, Y  +286.271, Z    +0.000, E1  +296.784, E3 -143914.297}
SPL {X   -98.696, Y  +256.580, Z    +0.000, E1  +308.006, E3 -144049.848}
ENDSPLINE

SPLINE
SPL {X  -138.661, Y  +302.689, Z    +0.000, E1  +316.811, E3 -144167.577}
SPL {X  -154.202, Y  +339.857, Z    +0.000, E1  +330.366, E3 -144185.230}
SPL {X  -158.556, Y  +361.128, Z    +0.000, E1  +342.470, E3 -144189.751}
SPL {X  -159.663, Y  +372.278, Z    +0.000, E1  +350.186, E3 -144191.033}
SPL {X  -159.986, Y  +381.388, Z    +0.000, E1  +357.201, E3 -144191.504}
SPL {X  -159.990, Y  +384.492, Z    +0.000, E1  +359.986, E3 -144191.554}
SPL {X  -159.990, Y  +385.649, Z    +0.000, E1  +361.559, E3 -144191.566}
SPL {X  -159.990, Y  +389.563, Z    +0.000, E1  +367.931, E3 -144191.698}
SPL {X  -159.990, Y  +396.421, Z    +0.000, E1  +380.831, E3 -144192.243}
SPL {X  -159.990, Y  +405.629, Z    +0.000, E1  +396.596, E3 -144193.598}
SPL {X  -159.990, Y  +417.919, Z    +0.000, E1  +410.108, E3 -144196.323}
SPL {X  -159.990, Y  +464.219, Z    +0.000, E1  +424.792, E3 -144214.382}
SPL {X  -159.990, Y  +601.948, Z    +0.000, E1  +428.261, E3 -144302.214}
SPL {X  -159.990, Y  +619.726, Z    +0.000, E1  +428.262, E3 -144317.275}
SPL {X  -159.990, Y  +636.530, Z    +0.000, E1  +428.257, E3 -144331.511}
SPL {X  -159.990, Y  +648.825, Z    +0.000, E1  +428.237, E3 -144341.970}
SPL {X  -159.990, Y  +661.441, Z    +0.000, E1  +428.256, E3 -144352.618}
SPL {X  -159.958, Y  +674.683, Z    +0.000, E1  +428.238, E3 -144363.881}
SPL {X  -159.269, Y  +686.675, Z    +0.000, E1  +428.163, E3 -144374.758}
SPL {X  -158.119, Y  +695.895, Z    +0.000, E1  +428.003, E3 -144383.799}
SPL {X  -156.550, Y  +704.498, Z    +0.000, E1  +427.821, E3 -144392.689}
SPL {X  -154.561, Y  +712.826, Z    +0.000, E1  +427.549, E3 -144401.820}
SPL {X  -152.048, Y  +721.282, Z    +0.000, E1  +427.243, E3 -144411.474}
SPL {X  -148.485, Y  +731.073, Z    +0.000, E1  +426.748, E3 -144423.324}
SPL {X  -145.075, Y  +738.953, Z    +0.000, E1  +426.252, E3 -144433.315}
SPL {X  -141.751, Y  +745.686, Z    +0.000, E1  +425.756, E3 -144442.146}
SPL {X  -138.928, Y  +750.847, Z    +0.000, E1  +425.305, E3 -144449.116}
SPL {X  -136.328, Y  +755.234, Z    +0.000, E1  +424.898, E3 -144455.106}
SPL {X  -132.717, Y  +760.848, Z    +0.000, E1  +424.322, E3 -144462.879}
SPL {X  -128.512, Y  +766.796, Z    +0.000, E1  +423.597, E3 -144471.234}
SPL {X   -99.023, Y  +797.163, Z    +0.000, E1  +413.965, E3 -144573.063}
ENDSPLINE

SPLINE
SPL {X  -130.021, Y  +764.727, Z    +0.000, E1  +405.990, E3 -144712.582}
SPL {X  -148.409, Y  +731.264, Z    +0.000, E1  +396.685, E3 -144736.296}
SPL {X  -155.017, Y  +711.078, Z    +0.000, E1  +387.846, E3 -144743.357}
SPL {X  -158.217, Y  +695.254, Z    +0.000, E1  +378.896, E3 -144746.800}
SPL {X  -159.762, Y  +680.037, Z    +0.000, E1  +368.585, E3 -144748.517}
SPL {X  -159.990, Y  +669.745, Z    +0.000, E1  +360.389, E3 -144748.939}
SPL {X  -159.990, Y  +666.879, Z    +0.000, E1  +356.292, E3 -144748.990}
SPL {X  -159.990, Y  +662.620, Z    +0.000, E1  +348.758, E3 -144749.191}
SPL {X  -159.990, Y  +657.714, Z    +0.000, E1  +339.502, E3 -144749.612}
SPL {X  -159.990, Y  +651.038, Z    +0.000, E1  +327.797, E3 -144750.515}
SPL {X  -159.990, Y  +637.243, Z    +0.000, E1  +311.500, E3 -144753.640}
SPL {X  -159.990, Y  +579.875, Z    +0.000, E1  +294.421, E3 -144776.499}
SPL {X  -159.990, Y  +453.091, Z    +0.000, E1  +291.862, E3 -144859.468}
SPL {X  -159.990, Y  +434.933, Z    +0.000, E1  +291.864, E3 -144874.962}
SPL {X  -159.990, Y  +420.071, Z    +0.000, E1  +291.886, E3 -144887.688}
SPL {X  -159.990, Y  +408.047, Z    +0.000, E1  +291.885, E3 -144897.935}
SPL {X  -159.990, Y  +395.904, Z    +0.000, E1  +291.881, E3 -144908.271}
SPL {X  -157.896, Y  +356.699, Z    +0.000, E1  +289.725, E3 -144920.581}
SPL {X  -156.475, Y  +349.148, Z    +0.000, E1  +290.612, E3 -144934.045}
SPL {X  -155.960, Y  +346.816, Z    +0.000, E1  +291.495, E3 -144943.206}
SPL {X  -154.913, Y  +342.515, Z    +0.000, E1  +292.501, E3 -144955.220}
SPL {X  -152.032, Y  +332.668, Z    +0.000, E1  +292.988, E3 -144967.211}
SPL {X  -148.460, Y  +322.864, Z    +0.000, E1  +293.452, E3 -144979.094}
SPL {X  -144.472, Y  +313.764, Z    +0.000, E1  +294.050, E3 -144990.757}
SPL {X  -141.765, Y  +308.342, Z    +0.000, E1  +294.475, E3 -144997.955}
SPL {X  -139.838, Y  +304.768, Z    +0.000, E1  +294.773, E3 -145002.774}
SPL {X  -137.162, Y  +300.138, Z    +0.000, E1  +295.180, E3 -145009.080}
SPL {X  -132.996, Y  +293.568, Z    +0.000, E1  +295.842, E3 -145018.215}
SPL {X  -128.628, Y  +287.360, Z    +0.000, E1  +296.617, E3 -145027.016}
SPL {X   -99.903, Y  +257.535, Z    +0.000, E1  +308.539, E3 -145175.879}
ENDSPLINE

SPLINE
SPL {X  -141.433, Y  +307.709, Z    +0.000, E1  +318.157, E3 -145285.676}
SPL {X  -151.246, Y  +330.333, Z    +0.000, E1  +326.099, E3 -145296.566}
SPL {X  -155.793, Y  +346.095, Z    +0.000, E1  +333.603, E3 -145301.225}
SPL {X  -158.556, Y  +361.128, Z    +0.000, E1  +342.470, E3 -145304.037}
SPL {X  -159.663, Y  +372.278, Z    +0.000, E1  +350.186, E3 -145305.319}
SPL {X  -159.986, Y  +381.388, Z    +0.000, E1  +357.201, E3 -145305.790}
SPL {X  -159.990, Y  +384.492, Z    +0.000, E1  +359.986, E3 -145305.840}
SPL {X  -159.990, Y  +385.649, Z    +0.000, E1  +361.559, E3 -145305.851}
SPL {X  -159.990, Y  +389.563, Z    +0.000, E1  +367.931, E3 -145305.984}
SPL {X  -159.990, Y  +396.421, Z    +0.000, E1  +380.831, E3 -145306.529}
SPL {X  -159.990, Y  +405.629, Z    +0.000, E1  +396.596, E3 -145307.883}
SPL {X  -159.990, Y  +418.631, Z    +0.000, E1  +410.627, E3 -145310.831}
SPL {X  -159.990, Y  +468.459, Z    +0.000, E1  +425.348, E3 -145330.374}
SPL {X  -159.990, Y  +601.948, Z    +0.000, E1  +428.261, E3 -145416.500}
SPL {X  -159.990, Y  +614.867, Z    +0.000, E1  +428.239, E3 -145427.498}
SPL {X  -159.990, Y  +627.954, Z    +0.000, E1  +428.256, E3 -145438.543}
SPL {X  -159.990, Y  +640.176, Z    +0.000, E1  +428.239, E3 -145448.922}
SPL {X  -159.990, Y  +653.116, Z    +0.000, E1  +428.255, E3 -145459.853}
SPL {X  -159.990, Y  +665.424, Z    +0.000, E1  +428.236, E3 -145470.318}
SPL {X  -159.958, Y  +674.683, Z    +0.000, E1  +428.238, E3 -145478.166}
SPL {X  -159.269, Y  +686.675, Z    +0.000, E1  +428.163, E3 -145489.044}
SPL {X  -158.119, Y  +695.895, Z    +0.000, E1  +428.003, E3 -145498.085}
SPL {X  -156.550, Y  +704.498, Z    +0.000, E1  +427.821, E3 -145506.975}
SPL {X  -153.468, Y  +716.715, Z    +0.000, E1  +427.444, E3 -145520.437}
SPL {X  -149.840, Y  +727.578, Z    +0.000, E1  +426.935, E3 -145533.313}
SPL {X  -145.768, Y  +737.444, Z    +0.000, E1  +426.379, E3 -145545.615}
SPL {X  -141.751, Y  +745.686, Z    +0.000, E1  +425.756, E3 -145556.432}
SPL {X  -138.928, Y  +750.847, Z    +0.000, E1  +425.305, E3 -145563.401}
SPL {X  -136.328, Y  +755.234, Z    +0.000, E1  +424.898, E3 -145569.392}
SPL {X  -132.717, Y  +760.848, Z    +0.000, E1  +424.322, E3 -145577.165}
SPL {X  -128.512, Y  +766.796, Z    +0.000, E1  +423.597, E3 -145585.519}
SPL {X   -99.023, Y  +797.163, Z    +0.000, E1  +413.965, E3 -145687.349}
ENDSPLINE

SPLINE
SPL {X  -130.021, Y  +764.727, Z    +0.000, E1  +405.990, E3 -145826.868}
SPL {X  -148.409, Y  +731.264, Z    +0.000, E1  +396.685, E3 -145850.582}
SPL {X  -155.017, Y  +711.078, Z    +0.000, E1  +387.846, E3 -145857.643}
SPL {X  -158.217, Y  +695.254, Z    +0.000, E1  +378.896, E3 -145861.086}
SPL {X  -159.524, Y  +683.703, Z    +0.000, E1  +371.166, E3 -145862.528}
SPL {X  -159.986, Y  +672.621, Z    +0.000, E1  +362.847, E3 -145863.169}
SPL {X  -159.990, Y  +669.426, Z    +0.000, E1  +359.932, E3 -145863.228}
SPL {X  -159.990, Y  +666.879, Z    +0.000, E1  +356.292, E3 -145863.276}
SPL {X  -159.990, Y  +662.620, Z    +0.000, E1  +348.758, E3 -145863.477}
SPL {X  -159.990, Y  +657.714, Z    +0.000, E1  +339.502, E3 -145863.898}
SPL {X  -159.990, Y  +651.038, Z    +0.000, E1  +327.797, E3 -145864.800}
SPL {X  -159.990, Y  +637.243, Z    +0.000, E1  +311.500, E3 -145867.926}
SPL {X  -159.990, Y  +579.875, Z    +0.000, E1  +294.421, E3 -145890.784}
SPL {X  -159.990, Y  +453.091, Z    +0.000, E1  +291.862, E3 -145973.754}
SPL {X  -159.990, Y  +434.933, Z    +0.000, E1  +291.864, E3 -145989.248}
SPL {X  -159.990, Y  +420.071, Z    +0.000, E1  +291.886, E3 -146001.974}
SPL {X  -159.990, Y  +408.047, Z    +0.000, E1  +291.885, E3 -146012.221}
SPL {X  -159.990, Y  +395.904, Z    +0.000, E1  +291.881, E3 -146022.557}
SPL {X  -157.896, Y  +356.699, Z    +0.000, E1  +289.725, E3 -146034.866}
SPL {X  -156.475, Y  +349.148, Z    +0.000, E1  +290.612, E3 -146048.330}
SPL {X  -155.960, Y  +346.816, Z    +0.000, E1  +291.495, E3 -146057.492}
SPL {X  -154.913, Y  +342.515, Z    +0.000, E1  +292.501, E3 -146069.506}
SPL {X  -152.032, Y  +332.668, Z    +0.000, E1  +292.988, E3 -146081.497}
SPL {X  -149.782, Y  +326.266, Z    +0.000, E1  +293.308, E3 -146089.237}
SPL {X  -146.798, Y  +318.884, Z    +0.000, E1  +293.699, E3 -146098.418}
SPL {X  -143.755, Y  +312.276, Z    +0.000, E1  +294.175, E3 -146107.027}
SPL {X  -140.755, Y  +306.442, Z    +0.000, E1  +294.606, E3 -146114.758}
SPL {X  -137.162, Y  +300.138, Z    +0.000, E1  +295.180, E3 -146123.366}
SPL {X  -134.303, Y  +295.555, Z    +0.000, E1  +295.659, E3 -146129.747}
SPL {X  -132.067, Y  +292.194, Z    +0.000, E1  +296.034, E3 -146134.479}
SPL {X  -128.628, Y  +287.360, Z    +0.000, E1  +296.617, E3 -146141.301}
SPL {X   -99.903, Y  +257.535, Z    +0.000, E1  +308.539, E3 -146290.164}
ENDSPLINE

SPLINE
SPL {X  -141.433, Y  +307.709, Z    +0.000, E1  +318.157, E3 -146399.961}
SPL {X  -151.246, Y  +330.333, Z    +0.000, E1  +326.099, E3 -146410.852}
SPL {X  -155.793, Y  +346.095, Z    +0.000, E1  +333.603, E3 -146415.510}
SPL {X  -158.556, Y  +361.128, Z    +0.000, E1  +342.470, E3 -146418.323}
SPL {X  -159.866, Y  +376.206, Z    +0.000, E1  +353.031, E3 -146419.852}
SPL {X  -159.990, Y  +384.326, Z    +0.000, E1  +359.760, E3 -146420.125}
SPL {X  -159.990, Y  +385.649, Z    +0.000, E1  +361.559, E3 -146420.137}
SPL {X  -159.990, Y  +389.563, Z    +0.000, E1  +367.931, E3 -146420.269}
SPL {X  -159.990, Y  +396.421, Z    +0.000, E1  +380.831, E3 -146420.814}
SPL {X  -159.990, Y  +405.629, Z    +0.000, E1  +396.596, E3 -146422.169}
SPL {X  -159.990, Y  +418.631, Z    +0.000, E1  +410.627, E3 -146425.116}
SPL {X  -159.990, Y  +468.459, Z    +0.000, E1  +425.348, E3 -146444.660}
SPL {X  -159.990, Y  +601.948, Z    +0.000, E1  +428.261, E3 -146530.786}
SPL {X  -159.990, Y  +619.726, Z    +0.000, E1  +428.262, E3 -146545.846}
SPL {X  -159.990, Y  +636.530, Z    +0.000, E1  +428.257, E3 -146560.083}
SPL {X  -159.990, Y  +653.116, Z    +0.000, E1  +428.255, E3 -146574.139}
SPL {X  -159.990, Y  +670.874, Z    +0.000, E1  +428.264, E3 -146589.154}
SPL {X  -159.269, Y  +686.675, Z    +0.000, E1  +428.163, E3 -146603.330}
SPL {X  -158.119, Y  +695.895, Z    +0.000, E1  +428.003, E3 -146612.370}
SPL {X  -156.550, Y  +704.498, Z    +0.000, E1  +427.821, E3 -146621.261}
SPL {X  -154.561, Y  +712.826, Z    +0.000, E1  +427.549, E3 -146630.391}
SPL {X  -152.048, Y  +721.282, Z    +0.000, E1  +427.243, E3 -146640.046}
SPL {X  -148.485, Y  +731.073, Z    +0.000, E1  +426.748, E3 -146651.895}
SPL {X  -145.075, Y  +738.953, Z    +0.000, E1  +426.252, E3 -146661.887}
SPL {X  -141.751, Y  +745.686, Z    +0.000, E1  +425.756, E3 -146670.718}
SPL {X  -138.928, Y  +750.847, Z    +0.000, E1  +425.305, E3 -146677.687}
SPL {X  -136.328, Y  +755.234, Z    +0.000, E1  +424.898, E3 -146683.677}
SPL {X  -132.717, Y  +760.848, Z    +0.000, E1  +424.322, E3 -146691.450}
SPL {X  -128.512, Y  +766.796, Z    +0.000, E1  +423.597, E3 -146699.805}
SPL {X   -99.023, Y  +797.163, Z    +0.000, E1  +413.965, E3 -146801.635}
ENDSPLINE

SPLINE
SPL {X  -130.021, Y  +764.727, Z    +0.000, E1  +405.990, E3 -146941.154}
SPL {X  -148.409, Y  +731.264, Z    +0.000, E1  +396.685, E3 -146964.867}
SPL {X  -155.017, Y  +711.078, Z    +0.000, E1  +387.846, E3 -146971.928}
SPL {X  -158.217, Y  +695.254, Z    +0.000, E1  +378.896, E3 -146975.371}
SPL {X  -159.762, Y  +680.037, Z    +0.000, E1  +368.585, E3 -146977.088}
SPL {X  -159.990, Y  +671.255, Z    +0.000, E1  +361.602, E3 -146977.494}
SPL {X  -159.990, Y  +669.426, Z    +0.000, E1  +359.932, E3 -146977.513}
SPL {X  -159.990, Y  +666.879, Z    +0.000, E1  +356.292, E3 -146977.561}
SPL {X  -159.990, Y  +662.620, Z    +0.000, E1  +348.758, E3 -146977.762}
SPL {X  -159.990, Y  +657.714, Z    +0.000, E1  +339.502, E3 -146978.184}
SPL {X  -159.990, Y  +651.038, Z    +0.000, E1  +327.797, E3 -146979.086}
SPL {X  -159.990, Y  +637.243, Z    +0.000, E1  +311.500, E3 -146982.211}
SPL {X  -159.990, Y  +579.875, Z    +0.000, E1  +294.421, E3 -147005.070}
SPL {X  -159.990, Y  +453.091, Z    +0.000, E1  +291.862, E3 -147088.039}
SPL {X  -159.990, Y  +434.933, Z    +0.000, E1  +291.864, E3 -147103.533}
SPL {X  -159.990, Y  +420.071, Z    +0.000, E1  +291.886, E3 -147116.259}
SPL {X  -159.990, Y  +408.047, Z    +0.000, E1  +291.885, E3 -147126.507}
SPL {X  -159.990, Y  +395.904, Z    +0.000, E1  +291.881, E3 -147136.843}
SPL {X  -158.518, Y  +360.846, Z    +0.000, E1  +289.610, E3 -147144.778}
SPL {X  -157.390, Y  +353.775, Z    +0.000, E1  +289.868, E3 -147152.454}
SPL {X  -156.475, Y  +349.148, Z    +0.000, E1  +290.612, E3 -147162.616}
SPL {X  -155.960, Y  +346.816, Z    +0.000, E1  +291.495, E3 -147171.777}
SPL {X  -154.913, Y  +342.515, Z    +0.000, E1  +292.501, E3 -147183.791}
SPL {X  -152.032, Y  +332.668, Z    +0.000, E1  +292.988, E3 -147195.783}
SPL {X  -149.782, Y  +326.266, Z    +0.000, E1  +293.308, E3 -147203.523}
SPL {X  -146.798, Y  +318.884, Z    +0.000, E1  +293.699, E3 -147212.703}
SPL {X  -143.755, Y  +312.276, Z    +0.000, E1  +294.175, E3 -147221.313}
SPL {X  -140.755, Y  +306.442, Z    +0.000, E1  +294.606, E3 -147229.044}
SPL {X  -137.162, Y  +300.138, Z    +0.000, E1  +295.180, E3 -147237.652}
SPL {X  -134.303, Y  +295.555, Z    +0.000, E1  +295.659, E3 -147244.033}
SPL {X  -132.067, Y  +292.194, Z    +0.000, E1  +296.034, E3 -147248.764}
SPL {X  -128.628, Y  +287.360, Z    +0.000, E1  +296.617, E3 -147255.587}
SPL {X   -98.696, Y  +256.580, Z    +0.000, E1  +308.006, E3 -147392.705}
ENDSPLINE

SPLINE
SPL {X  -138.661, Y  +302.689, Z    +0.000, E1  +316.811, E3 -147510.434}
SPL {X  -154.202, Y  +339.857, Z    +0.000, E1  +330.366, E3 -147528.087}
SPL {X  -158.556, Y  +361.128, Z    +0.000, E1  +342.470, E3 -147532.609}
SPL {X  -159.866, Y  +376.206, Z    +0.000, E1  +353.031, E3 -147534.138}
SPL {X  -159.990, Y  +384.789, Z    +0.000, E1  +360.146, E3 -147534.415}
SPL {X  -159.990, Y  +388.306, Z    +0.000, E1  +365.901, E3 -147534.494}
SPL {X  -159.990, Y  +392.624, Z    +0.000, E1  +373.655, E3 -147534.744}
SPL {X  -159.990, Y  +398.511, Z    +0.000, E1  +384.979, E3 -147535.324}
SPL {X  -159.990, Y  +405.629, Z    +0.000, E1  +396.596, E3 -147536.455}
SPL {X  -159.990, Y  +418.631, Z    +0.000, E1  +410.627, E3 -147539.402}
SPL {X  -159.990, Y  +468.459, Z    +0.000, E1  +425.348, E3 -147558.945}
SPL {X  -159.990, Y  +601.948, Z    +0.000, E1  +428.261, E3 -147645.071}
SPL {X  -159.990, Y  +614.867, Z    +0.000, E1  +428.239, E3 -147656.070}
SPL {X  -159.990, Y  +627.954, Z    +0.000, E1  +428.256, E3 -147667.114}
SPL {X  -159.990, Y  +640.176, Z    +0.000, E1  +428.239, E3 -147677.493}
SPL {X  -159.990, Y  +653.116, Z    +0.000, E1  +428.255, E3 -147688.425}
SPL {X  -159.990, Y  +665.424, Z    +0.000, E1  +428.236, E3 -147698.889}
SPL {X  -159.958, Y  +674.683, Z    +0.000, E1  +428.238, E3 -147706.738}
SPL {X  -159.269, Y  +686.675, Z    +0.000, E1  +428.163, E3 -147717.615}
SPL {X  -157.606, Y  +699.018, Z    +0.000, E1  +427.957, E3 -147729.799}
SPL {X  -155.210, Y  +710.317, Z    +0.000, E1  +427.656, E3 -147741.839}
SPL {X  -152.683, Y  +719.299, Z    +0.000, E1  +427.307, E3 -147752.051}
SPL {X  -149.840, Y  +727.578, Z    +0.000, E1  +426.935, E3 -147761.885}
SPL {X  -145.768, Y  +737.444, Z    +0.000, E1  +426.379, E3 -147774.187}
SPL {X  -141.751, Y  +745.686, Z    +0.000, E1  +425.756, E3 -147785.003}
SPL {X  -138.928, Y  +750.847, Z    +0.000, E1  +425.305, E3 -147791.973}
SPL {X  -136.328, Y  +755.234, Z    +0.000, E1  +424.898, E3 -147797.963}
SPL {X  -132.717, Y  +760.848, Z    +0.000, E1  +424.322, E3 -147805.736}
SPL {X  -129.778, Y  +765.065, Z    +0.000, E1  +423.787, E3 -147811.691}
SPL {X  -127.600, Y  +768.014, Z    +0.000, E1  +423.408, E3 -147815.838}
SPL {X   -99.023, Y  +797.163, Z    +0.000, E1  +413.965, E3 -147915.920}
ENDSPLINE

SPLINE
SPL {X  -130.021, Y  +764.727, Z    +0.000, E1  +405.990, E3 -148055.440}
SPL {X  -148.409, Y  +731.264, Z    +0.000, E1  +396.685, E3 -148079.153}
SPL {X  -155.017, Y  +711.078, Z    +0.000, E1  +387.846, E3 -148086.214}
SPL {X  -158.217, Y  +695.254, Z    +0.000, E1  +378.896, E3 -148089.657}
SPL {X  -159.524, Y  +683.703, Z    +0.000, E1  +371.166, E3 -148091.099}
SPL {X  -159.986, Y  +672.621, Z    +0.000, E1  +362.847, E3 -148091.741}
SPL {X  -159.990, Y  +669.148, Z    +0.000, E1  +359.679, E3 -148091.802}
SPL {X  -159.990, Y  +666.130, Z    +0.000, E1  +354.946, E3 -148091.868}
SPL {X  -159.990, Y  +662.620, Z    +0.000, E1  +348.758, E3 -148092.048}
SPL {X  -159.990, Y  +657.714, Z    +0.000, E1  +339.502, E3 -148092.469}
SPL {X  -159.990, Y  +651.038, Z    +0.000, E1  +327.797, E3 -148093.372}
SPL {X  -159.990, Y  +637.243, Z    +0.000, E1  +311.500, E3 -148096.497}
SPL {X  -159.990, Y  +579.875, Z    +0.000, E1  +294.421, E3 -148119.356}
SPL {X  -159.990, Y  +453.091, Z    +0.000, E1  +291.862, E3 -148202.325}
SPL {X  -159.990, Y  +434.933, Z    +0.000, E1  +291.864, E3 -148217.819}
SPL {X  -159.990, Y  +420.071, Z    +0.000, E1  +291.886, E3 -148230.545}
SPL {X  -159.990, Y  +408.047, Z    +0.000, E1  +291.885, E3 -148240.792}
SPL {X  -159.990, Y  +395.904, Z    +0.000, E1  +291.881, E3 -148251.128}
SPL {X  -157.896, Y  +356.699, Z    +0.000, E1  +289.725, E3 -148263.438}
SPL {X  -156.475, Y  +349.148, Z    +0.000, E1  +290.612, E3 -148276.902}
SPL {X  -155.786, Y  +346.063, Z    +0.000, E1  +291.892, E3 -148290.196}
SPL {X  -153.671, Y  +337.981, Z    +0.000, E1  +292.746, E3 -148303.816}
SPL {X  -150.407, Y  +327.960, Z    +0.000, E1  +293.203, E3 -148315.705}
SPL {X  -146.798, Y  +318.884, Z    +0.000, E1  +293.699, E3 -148326.989}
SPL {X  -142.741, Y  +310.238, Z    +0.000, E1  +294.301, E3 -148338.248}
SPL {X  -139.838, Y  +304.768, Z    +0.000, E1  +294.773, E3 -148345.631}
SPL {X  -137.162, Y  +300.138, Z    +0.000, E1  +295.180, E3 -148351.937}
SPL {X  -132.996, Y  +293.568, Z    +0.000, E1  +295.842, E3 -148361.072}
SPL {X  -128.628, Y  +287.360, Z    +0.000, E1  +296.617, E3 -148369.873}
SPL {X   -98.696, Y  +256.580, Z    +0.000, E1  +308.006, E3 -148506.991}
ENDSPLINE

SPLINE
SPL {X  -138.661, Y  +302.689, Z    +0.000, E1  +316.811, E3 -148624.720}
SPL {X  -154.202, Y  +339.857, Z    +0.000, E1  +330.366, E3 -148642.373}
SPL {X  -158.556, Y  +361.128, Z    +0.000, E1  +342.470, E3 -148646.894}
SPL {X  -159.866, Y  +376.206, Z    +0.000, E1  +353.031, E3 -148648.423}
SPL {X  -159.990, Y  +384.789, Z    +0.000, E1  +360.146, E3 -148648.700}
SPL {X  -159.990, Y  +388.306, Z    +0.000, E1  +365.901, E3 -148648.780}
SPL {X  -159.990, Y  +392.624, Z    +0.000, E1  +373.655, E3 -148649.029}
SPL {X  -159.990, Y  +398.511, Z    +0.000, E1  +384.979, E3 -148649.610}
SPL {X  -159.990, Y  +405.629, Z    +0.000, E1  +396.596, E3 -148650.740}
SPL {X  -159.990, Y  +417.919, Z    +0.000, E1  +410.108, E3 -148653.466}
SPL {X  -159.990, Y  +464.219, Z    +0.000, E1  +424.792, E3 -148671.525}
SPL {X  -159.990, Y  +601.948, Z    +0.000, E1  +428.261, E3 -148759.357}
SPL {X  -159.990, Y  +614.867, Z    +0.000, E1  +428.239, E3 -148770.356}
SPL {X  -159.990, Y  +627.954, Z    +0.000, E1  +428.256, E3 -148781.400}
SPL {X  -159.990, Y  +640.176, Z    +0.000, E1  +428.239, E3 -148791.779}
SPL {X  -159.990, Y  +653.116, Z    +0.000, E1  +428.255, E3 -148802.710}
SPL {X  -159.990, Y  +665.424, Z    +0.000, E1  +428.236, E3 -148813.175}
SPL {X  -159.958, Y  +674.683, Z    +0.000, E1  +428.238, E3 -148821.024}
SPL {X  -159.269, Y  +686.675, Z    +0.000, E1  +428.163, E3 -148831.901}
SPL {X  -158.119, Y  +695.895, Z    +0.000, E1  +428.003, E3 -148840.942}
SPL {X  -156.550, Y  +704.498, Z    +0.000, E1  +427.821, E3 -148849.832}
SPL {X  -153.468, Y  +716.715, Z    +0.000, E1  +427.444, E3 -148863.295}
SPL {X  -149.089, Y  +729.545, Z    +0.000, E1  +426.860, E3 -148878.528}
SPL {X  -145.075, Y  +738.953, Z    +0.000, E1  +426.252, E3 -148890.458}
SPL {X  -141.751, Y  +745.686, Z    +0.000, E1  +425.756, E3 -148899.289}
SPL {X  -138.928, Y  +750.847, Z    +0.000, E1  +425.305, E3 -148906.258}
SPL {X  -135.390, Y  +756.743, Z    +0.000, E1  +424.775, E3 -148914.290}
SPL {X  -132.002, Y  +761.900, Z    +0.000, E1  +424.179, E3 -148921.522}
SPL {X  -128.512, Y  +766.796, Z    +0.000, E1  +423.597, E3 -148928.376}
SPL {X   -99.023, Y  +797.163, Z    +0.000, E1  +413.965, E3 -149030.206}
ENDSPLINE

SPLINE
SPL {X  -130.021, Y  +764.727, Z    +0.000, E1  +405.990, E3 -149169.725}
SPL {X  -148.409, Y  +731.264, Z    +0.000, E1  +396.685, E3 -149193.439}
SPL {X  -155.017, Y  +711.078, Z    +0.000, E1  +387.846, E3 -149200.500}
SPL {X  -158.217, Y  +695.254, Z    +0.000, E1  +378.896, E3 -149203.943}
SPL {X  -159.524, Y  +683.703, Z    +0.000, E1  +371.166, E3 -149205.385}
SPL {X  -159.986, Y  +672.621, Z    +0.000, E1  +362.847, E3 -149206.026}
SPL {X  -159.990, Y  +669.148, Z    +0.000, E1  +359.679, E3 -149206.088}
SPL {X  -159.990, Y  +666.130, Z    +0.000, E1  +354.946, E3 -149206.154}
SPL {X  -159.990, Y  +662.620, Z    +0.000, E1  +348.758, E3 -149206.334}
SPL {X  -159.990, Y  +657.714, Z    +0.000, E1  +339.502, E3 -149206.755}
SPL {X  -159.990, Y  +651.038, Z    +0.000, E1  +327.797, E3 -149207.658}
SPL {X  -159.990, Y  +637.243, Z    +0.000, E1  +311.500, E3 -149210.783}
SPL {X  -159.990, Y  +579.875, Z    +0.000, E1  +294.421, E3 -149233.641}
SPL {X  -159.990, Y  +453.091, Z    +0.000, E1  +291.862, E3 -149316.611}
SPL {X  -159.990, Y  +434.933, Z    +0.000, E1  +291.864, E3 -149332.105}
SPL {X  -159.990, Y  +420.071, Z    +0.000, E1  +291.886, E3 -149344.831}
SPL {X  -159.990, Y  +408.047, Z    +0.000, E1  +291.885, E3 -149355.078}
SPL {X  -159.990, Y  +395.904, Z    +0.000, E1  +291.881, E3 -149365.414}
SPL {X  -157.896, Y  +356.699, Z    +0.000, E1  +289.725, E3 -149377.724}
SPL {X  -156.475, Y  +349.148, Z    +0.000, E1  +290.612, E3 -149391.188}
SPL {X  -155.960, Y  +346.816, Z    +0.000, E1  +291.495, E3 -149400.349}
SPL {X  -154.913, Y  +342.515, Z    +0.000, E1  +292.501, E3 -149412.363}
SPL {X  -152.032, Y  +332.668, Z    +0.000, E1  +292.988, E3 -149424.354}
SPL {X  -149.782, Y  +326.266, Z    +0.000, E1  +293.308, E3 -149432.094}
SPL {X  -146.798, Y  +318.884, Z    +0.000, E1  +293.699, E3 -149441.275}
SPL {X  -143.755, Y  +312.276, Z    +0.000, E1  +294.175, E3 -149449.884}
SPL {X  -140.755, Y  +306.442, Z    +0.000, E1  +294.606, E3 -149457.615}
SPL {X  -137.162, Y  +300.138, Z    +0.000, E1  +295.180, E3 -149466.223}
SPL {X  -134.303, Y  +295.555, Z    +0.000, E1  +295.659, E3 -149472.604}
SPL {X  -132.067, Y  +292.194, Z    +0.000, E1  +296.034, E3 -149477.336}
SPL {X  -128.628, Y  +287.360, Z    +0.000, E1  +296.617, E3 -149484.159}
SPL {X   -98.696, Y  +256.580, Z    +0.000, E1  +308.006, E3 -149621.277}
ENDSPLINE

SPLINE
SPL {X  -138.661, Y  +302.689, Z    +0.000, E1  +316.811, E3 -149739.005}
SPL {X  -154.202, Y  +339.857, Z    +0.000, E1  +330.366, E3 -149756.658}
SPL {X  -158.556, Y  +361.128, Z    +0.000, E1  +342.470, E3 -149761.180}
SPL {X  -159.866, Y  +376.206, Z    +0.000, E1  +353.031, E3 -149762.709}
SPL {X  -159.990, Y  +384.326, Z    +0.000, E1  +359.760, E3 -149762.982}
SPL {X  -159.990, Y  +385.649, Z    +0.000, E1  +361.559, E3 -149762.994}
SPL {X  -159.990, Y  +388.306, Z    +0.000, E1  +365.901, E3 -149763.066}
SPL {X  -159.990, Y  +392.624, Z    +0.000, E1  +373.655, E3 -149763.315}
SPL {X  -159.990, Y  +398.511, Z    +0.000, E1  +384.979, E3 -149763.895}
SPL {X  -159.990, Y  +405.629, Z    +0.000, E1  +396.596, E3 -149765.026}
SPL {X  -159.990, Y  +418.631, Z    +0.000, E1  +410.627, E3 -149767.973}
SPL {X  -159.990, Y  +468.459, Z    +0.000, E1  +425.348, E3 -149787.517}
SPL {X  -159.990, Y  +601.948, Z    +0.000, E1  +428.261, E3 -149873.643}
SPL {X  -159.990, Y  +619.726, Z    +0.000, E1  +428.262, E3 -149888.704}
SPL {X  -159.990, Y  +636.530, Z    +0.000, E1  +428.257, E3 -149902.940}
SPL {X  -159.990, Y  +653.116, Z    +0.000, E1  +428.255, E3 -149916.996}
SPL {X  -159.990, Y  +670.874, Z    +0.000, E1  +428.264, E3 -149932.011}
SPL {X  -159.269, Y  +686.675, Z    +0.000, E1  +428.163, E3 -149946.187}
SPL {X  -157.606, Y  +699.018, Z    +0.000, E1  +427.957, E3 -149958.370}
SPL {X  -155.210, Y  +710.317, Z    +0.000, E1  +427.656, E3 -149970.410}
SPL {X  -152.048, Y  +721.282, Z    +0.000, E1  +427.243, E3 -149982.903}
SPL {X  -148.485, Y  +731.073, Z    +0.000, E1  +426.748, E3 -149994.752}
SPL {X  -145.075, Y  +738.953, Z    +0.000, E1  +426.252, E3 -150004.744}
SPL {X  -141.751, Y  +745.686, Z    +0.000, E1  +425.756, E3 -150013.575}
SPL {X  -138.928, Y  +750.847, Z    +0.000, E1  +425.305, E3 -150020.544}
SPL {X  -136.328, Y  +755.234, Z    +0.000, E1  +424.898, E3 -150026.534}
SPL {X  -132.717, Y  +760.848, Z    +0.000, E1  +424.322, E3 -150034.308}
SPL {X  -128.512, Y  +766.796, Z    +0.000, E1  +423.597, E3 -150042.662}
SPL {X   -99.023, Y  +797.163, Z    +0.000, E1  +413.965, E3 -150144.492}
ENDSPLINE

SPLINE
SPL {X  -130.021, Y  +764.727, Z    +0.000, E1  +405.990, E3 -150284.011}
SPL {X  -148.409, Y  +731.264, Z    +0.000, E1  +396.685, E3 -150307.725}
SPL {X  -155.017, Y  +711.078, Z    +0.000, E1  +387.846, E3 -150314.786}
SPL {X  -158.217, Y  +695.254, Z    +0.000, E1  +378.896, E3 -150318.228}
SPL {X  -159.762, Y  +680.037, Z    +0.000, E1  +368.585, E3 -150319.945}
SPL {X  -159.990, Y  +671.255, Z    +0.000, E1  +361.602, E3 -150320.351}
SPL {X  -159.990, Y  +669.426, Z    +0.000, E1  +359.932, E3 -150320.371}
SPL {X  -159.990, Y  +666.879, Z    +0.000, E1  +356.292, E3 -150320.418}
SPL {X  -159.990, Y  +662.620, Z    +0.000, E1  +348.758, E3 -150320.620}
SPL {X  -159.990, Y  +657.714, Z    +0.000, E1  +339.502, E3 -150321.041}
SPL {X  -159.990, Y  +651.038, Z    +0.000, E1  +327.797, E3 -150321.943}
SPL {X  -159.990, Y  +637.243, Z    +0.000, E1  +311.500, E3 -150325.068}
SPL {X  -159.990, Y  +579.875, Z    +0.000, E1  +294.421, E3 -150347.927}
SPL {X  -159.990, Y  +453.091, Z    +0.000, E1  +291.862, E3 -150430.897}
SPL {X  -159.990, Y  +434.933, Z    +0.000, E1  +291.864, E3 -150446.390}
SPL {X  -159.990, Y  +420.071, Z    +0.000, E1  +291.886, E3 -150459.116}
SPL {X  -159.990, Y  +408.047, Z    +0.000, E1  +291.885, E3 -150469.364}
SPL {X  -159.990, Y  +395.904, Z    +0.000, E1  +291.881, E3 -150479.700}
SPL {X  -157.896, Y  +356.699, Z    +0.000, E1  +289.725, E3 -150492.009}
SPL {X  -156.475, Y  +349.148, Z    +0.000, E1  +290.612, E3 -150505.473}
SPL {X  -155.960, Y  +346.816, Z    +0.000, E1  +291.495, E3 -150514.635}
SPL {X  -154.913, Y  +342.515, Z    +0.000, E1  +292.501, E3 -150526.649}
SPL {X  -152.032, Y  +332.668, Z    +0.000, E1  +292.988, E3 -150538.640}
SPL {X  -148.460, Y  +322.864, Z    +0.000, E1  +293.452, E3 -150550.523}
SPL {X  -144.472, Y  +313.764, Z    +0.000, E1  +294.050, E3 -150562.186}
SPL {X  -140.755, Y  +306.442, Z    +0.000, E1  +294.606, E3 -150571.901}
SPL {X  -137.162, Y  +300.138, Z    +0.000, E1  +295.180, E3 -150580.509}
SPL {X  -134.303, Y  +295.555, Z    +0.000, E1  +295.659, E3 -150586.890}
SPL {X  -131.069, Y  +290.753, Z    +0.000, E1  +296.178, E3 -150593.623}
SPL {X  -127.815, Y  +286.271, Z    +0.000, E1  +296.784, E3 -150600.012}
SPL {X   -98.696, Y  +256.580, Z    +0.000, E1  +308.006, E3 -150735.562}
ENDSPLINE

SPLINE
SPL {X  -138.661, Y  +302.689, Z    +0.000, E1  +316.811, E3 -150853.291}
SPL {X  -154.202, Y  +339.857, Z    +0.000, E1  +330.366, E3 -150870.944}
SPL {X  -158.556, Y  +361.128, Z    +0.000, E1  +342.470, E3 -150875.466}
SPL {X  -159.663, Y  +372.278, Z    +0.000, E1  +350.186, E3 -150876.747}
SPL {X  -159.986, Y  +381.388, Z    +0.000, E1  +357.201, E3 -150877.218}
SPL {X  -159.990, Y  +384.492, Z    +0.000, E1  +359.986, E3 -150877.269}
SPL {X  -159.990, Y  +385.649, Z    +0.000, E1  +361.559, E3 -150877.280}
SPL {X  -159.990, Y  +389.563, Z    +0.000, E1  +367.931, E3 -150877.412}
SPL {X  -159.990, Y  +396.421, Z    +0.000, E1  +380.831, E3 -150877.957}
SPL {X  -159.990, Y  +405.629, Z    +0.000, E1  +396.596, E3 -150879.312}
SPL {X  -159.990, Y  +418.631, Z    +0.000, E1  +410.627, E3 -150882.259}
SPL {X  -159.990, Y  +468.459, Z    +0.000, E1  +425.348, E3 -150901.803}
SPL {X  -159.990, Y  +601.948, Z    +0.000, E1  +428.261, E3 -150987.929}
SPL {X  -159.990, Y  +619.726, Z    +0.000, E1  +428.262, E3 -151002.989}
SPL {X  -159.990, Y  +636.530, Z    +0.000, E1  +428.257, E3 -151017.225}
SPL {X  -159.990, Y  +648.825, Z    +0.000, E1  +428.237, E3 -151027.684}
SPL {X  -159.990, Y  +661.441, Z    +0.000, E1  +428.256, E3 -151038.332}
SPL {X  -159.958, Y  +674.683, Z    +0.000, E1  +428.238, E3 -151049.595}
SPL {X  -159.269, Y  +686.675, Z    +0.000, E1  +428.163, E3 -151060.472}
SPL {X  -157.606, Y  +699.018, Z    +0.000, E1  +427.957, E3 -151072.656}
SPL {X  -155.210, Y  +710.317, Z    +0.000, E1  +427.656, E3 -151084.696}
SPL {X  -152.048, Y  +721.282, Z    +0.000, E1  +427.243, E3 -151097.189}
SPL {X  -148.485, Y  +731.073, Z    +0.000, E1  +426.748, E3 -151109.038}
SPL {X  -145.075, Y  +738.953, Z    +0.000, E1  +426.252, E3 -151119.029}
SPL {X  -141.751, Y  +745.686, Z    +0.000, E1  +425.756, E3 -151127.860}
SPL {X  -138.928, Y  +750.847, Z    +0.000, E1  +425.305, E3 -151134.830}
SPL {X  -136.328, Y  +755.234, Z    +0.000, E1  +424.898, E3 -151140.820}
SPL {X  -132.717, Y  +760.848, Z    +0.000, E1  +424.322, E3 -151148.593}
SPL {X  -128.512, Y  +766.796, Z    +0.000, E1  +423.597, E3 -151156.948}
SPL {X   -99.023, Y  +797.163, Z    +0.000, E1  +413.965, E3 -151258.777}
ENDSPLINE

SPLINE
SPL {X  -130.021, Y  +764.727, Z    +0.000, E1  +405.990, E3 -151398.297}
SPL {X  -148.409, Y  +731.264, Z    +0.000, E1  +396.685, E3 -151422.010}
SPL {X  -155.017, Y  +711.078, Z    +0.000, E1  +387.846, E3 -151429.071}
SPL {X  -158.217, Y  +695.254, Z    +0.000, E1  +378.896, E3 -151432.514}
SPL {X  -159.762, Y  +680.037, Z    +0.000, E1  +368.585, E3 -151434.231}
SPL {X  -159.990, Y  +671.255, Z    +0.000, E1  +361.602, E3 -151434.637}
SPL {X  -159.990, Y  +669.426, Z    +0.000, E1  +359.932, E3 -151434.656}
SPL {X  -159.990, Y  +666.879, Z    +0.000, E1  +356.292, E3 -151434.704}
SPL {X  -159.990, Y  +662.620, Z    +0.000, E1  +348.758, E3 -151434.905}
SPL {X  -159.990, Y  +657.714, Z    +0.000, E1  +339.502, E3 -151435.327}
SPL {X  -159.990, Y  +651.038, Z    +0.000, E1  +327.797, E3 -151436.229}
SPL {X  -159.990, Y  +637.243, Z    +0.000, E1  +311.500, E3 -151439.354}
SPL {X  -159.990, Y  +579.875, Z    +0.000, E1  +294.421, E3 -151462.213}
SPL {X  -159.990, Y  +453.091, Z    +0.000, E1  +291.862, E3 -151545.182}
SPL {X  -159.990, Y  +434.933, Z    +0.000, E1  +291.864, E3 -151560.676}
SPL {X  -159.990, Y  +420.071, Z    +0.000, E1  +291.886, E3 -151573.402}
SPL {X  -159.990, Y  +408.047, Z    +0.000, E1  +291.885, E3 -151583.650}
SPL {X  -159.990, Y  +395.904, Z    +0.000, E1  +291.881, E3 -151593.986}
SPL {X  -157.896, Y  +356.699, Z    +0.000, E1  +289.725, E3 -151606.295}
SPL {X  -156.475, Y  +349.148, Z    +0.000, E1  +290.612, E3 -151619.759}
SPL {X  -155.786, Y  +346.063, Z    +0.000, E1  +291.892, E3 -151633.053}
SPL {X  -153.671, Y  +337.981, Z    +0.000, E1  +292.746, E3 -151646.673}
SPL {X  -150.407, Y  +327.960, Z    +0.000, E1  +293.203, E3 -151658.562}
SPL {X  -146.798, Y  +318.884, Z    +0.000, E1  +293.699, E3 -151669.846}
SPL {X  -142.741, Y  +310.238, Z    +0.000, E1  +294.301, E3 -151681.105}
SPL {X  -139.838, Y  +304.768, Z    +0.000, E1  +294.773, E3 -151688.488}
SPL {X  -137.162, Y  +300.138, Z    +0.000, E1  +295.180, E3 -151694.795}
SPL {X  -132.996, Y  +293.568, Z    +0.000, E1  +295.842, E3 -151703.929}
SPL {X  -128.628, Y  +287.360, Z    +0.000, E1  +296.617, E3 -151712.730}
SPL {X   -98.696, Y  +256.580, Z    +0.000, E1  +308.006, E3 -151849.848}
ENDSPLINE

SPLINE
SPL {X  -138.661, Y  +302.689, Z    +0.000, E1  +316.811, E3 -151967.577}
SPL {X  -151.246, Y  +330.333, Z    +0.000, E1  +326.099, E3 -151982.281}
SPL {X  -155.793, Y  +346.095, Z    +0.000, E1  +333.603, E3 -151986.939}
SPL {X  -158.556, Y  +361.128, Z    +0.000, E1  +342.470, E3 -151989.751}
SPL {X  -159.663, Y  +372.278, Z    +0.000, E1  +350.186, E3 -151991.033}
SPL {X  -159.986, Y  +381.388, Z    +0.000, E1  +357.201, E3 -151991.504}
SPL {X  -159.990, Y  +384.492, Z    +0.000, E1  +359.986, E3 -151991.554}
SPL {X  -159.990, Y  +385.649, Z    +0.000, E1  +361.559, E3 -151991.566}
SPL {X  -159.990, Y  +388.306, Z    +0.000, E1  +365.901, E3 -151991.637}
SPL {X  -159.990, Y  +392.624, Z    +0.000, E1  +373.655, E3 -151991.887}
SPL {X  -159.990, Y  +398.511, Z    +0.000, E1  +384.979, E3 -151992.467}
SPL {X  -159.990, Y  +405.629, Z    +0.000, E1  +396.596, E3 -151993.598}
SPL {X  -159.990, Y  +418.631, Z    +0.000, E1  +410.627, E3 -151996.545}
SPL {X  -159.990, Y  +468.459, Z    +0.000, E1  +425.348, E3 -152016.088}
SPL {X  -159.990, Y  +601.948, Z    +0.000, E1  +428.261, E3 -152102.214}
SPL {X  -159.990, Y  +614.867, Z    +0.000, E1  +428.239, E3 -152113.213}
SPL {X  -159.990, Y  +627.954, Z    +0.000, E1  +428.256, E3 -152124.257}
SPL {X  -159.990, Y  +640.176, Z    +0.000, E1  +428.239, E3 -152134.636}
SPL {X  -159.990, Y  +653.116, Z    +0.000, E1  +428.255, E3 -152145.568}
SPL {X  -159.990, Y  +670.874, Z    +0.000, E1  +428.264, E3 -152160.582}
SPL {X  -159.269, Y  +686.675, Z    +0.000, E1  +428.163, E3 -152174.758}
SPL {X  -158.119, Y  +695.895, Z    +0.000, E1  +428.003, E3 -152183.799}
SPL {X  -156.550, Y  +704.498, Z    +0.000, E1  +427.821, E3 -152192.689}
SPL {X  -153.468, Y  +716.715, Z    +0.000, E1  +427.444, E3 -152206.152}
SPL {X  -149.840, Y  +727.578, Z    +0.000, E1  +426.935, E3 -152219.028}
SPL {X  -145.768, Y  +737.444, Z    +0.000, E1  +426.379, E3 -152231.330}
SPL {X  -141.751, Y  +745.686, Z    +0.000, E1  +425.756, E3 -152242.146}
SPL {X  -138.928, Y  +750.847, Z    +0.000, E1  +425.305, E3 -152249.116}
SPL {X  -136.328, Y  +755.234, Z    +0.000, E1  +424.898, E3 -152255.106}
SPL {X  -132.717, Y  +760.848, Z    +0.000, E1  +424.322, E3 -152262.879}
SPL {X  -128.512, Y  +766.796, Z    +0.000, E1  +423.597, E3 -152271.234}
SPL {X   -99.023, Y  +797.163, Z    +0.000, E1  +413.965, E3 -152373.063}
ENDSPLINE

SPLINE
SPL {X  -130.021, Y  +764.727, Z    +0.000, E1  +405.990, E3 -152512.582}
SPL {X  -148.409, Y  +731.264, Z    +0.000, E1  +396.685, E3 -152536.296}
SPL {X  -155.017, Y  +711.078, Z    +0.000, E1  +387.846, E3 -152543.357}
SPL {X  -158.217, Y  +695.254, Z    +0.000, E1  +378.896, E3 -152546.800}
SPL {X  -159.762, Y  +680.037, Z    +0.000, E1  +368.585, E3 -152548.517}
SPL {X  -159.990, Y  +671.255, Z    +0.000, E1  +361.602, E3 -152548.922}
SPL {X  -159.990, Y  +669.426, Z    +0.000, E1  +359.932, E3 -152548.942}
SPL {X  -159.990, Y  +666.879, Z    +0.000, E1  +356.292, E3 -152548.990}
SPL {X  -159.990, Y  +662.620, Z    +0.000, E1  +348.758, E3 -152549.191}
SPL {X  -159.990, Y  +657.714, Z    +0.000, E1  +339.502, E3 -152549.612}
SPL {X  -159.990, Y  +651.038, Z    +0.000, E1  +327.797, E3 -152550.515}
SPL {X  -159.990, Y  +642.324, Z    +0.000, E1  +316.129, E3 -152552.249}
SPL {X  -159.990, Y  +634.003, Z    +0.000, E1  +308.893, E3 -152554.525}
SPL {X  -159.990, Y  +579.875, Z    +0.000, E1  +294.421, E3 -152576.499}
SPL {X  -159.990, Y  +453.091, Z    +0.000, E1  +291.862, E3 -152659.468}
SPL {X  -159.990, Y  +434.933, Z    +0.000, E1  +291.864, E3 -152674.962}
SPL {X  -159.990, Y  +420.071, Z    +0.000, E1  +291.886, E3 -152687.688}
SPL {X  -159.990, Y  +408.047, Z    +0.000, E1  +291.885, E3 -152697.935}
SPL {X  -159.990, Y  +395.904, Z    +0.000, E1  +291.881, E3 -152708.271}
SPL {X  -157.896, Y  +356.699, Z    +0.000, E1  +289.725, E3 -152720.581}
SPL {X  -156.475, Y  +349.148, Z    +0.000, E1  +290.612, E3 -152734.045}
SPL {X  -155.960, Y  +346.816, Z    +0.000, E1  +291.495, E3 -152743.206}
SPL {X  -154.913, Y  +342.515, Z    +0.000, E1  +292.501, E3 -152755.220}
SPL {X  -152.032, Y  +332.668, Z    +0.000, E1  +292.988, E3 -152767.211}
SPL {X  -149.782, Y  +326.266, Z    +0.000, E1  +293.308, E3 -152774.951}
SPL {X  -146.798, Y  +318.884, Z    +0.000, E1  +293.699, E3 -152784.132}
SPL {X  -143.755, Y  +312.276, Z    +0.000, E1  +294.175, E3 -152792.741}
SPL {X  -140.755, Y  +306.442, Z    +0.000, E1  +294.606, E3 -152800.472}
SPL {X  -137.162, Y  +300.138, Z    +0.000, E1  +295.180, E3 -152809.080}
SPL {X  -134.303, Y  +295.555, Z    +0.000, E1  +295.659, E3 -152815.461}
SPL {X  -132.067, Y  +292.194, Z    +0.000, E1  +296.034, E3 -152820.193}
SPL {X  -128.628, Y  +287.360, Z    +0.000, E1  +296.617, E3 -152827.016}
SPL {X   -99.903, Y  +257.535, Z    +0.000, E1  +308.539, E3 -152975.879}
ENDSPLINE

SPLINE
SPL {X  -141.433, Y  +307.709, Z    +0.000, E1  +318.157, E3 -153085.676}
SPL {X  -151.246, Y  +330.333, Z    +0.000, E1  +326.099, E3 -153096.566}
SPL {X  -155.793, Y  +346.095, Z    +0.000, E1  +333.603, E3 -153101.225}
SPL {X  -158.556, Y  +361.128, Z    +0.000, E1  +342.470, E3 -153104.037}
SPL {X  -159.866, Y  +376.206, Z    +0.000, E1  +353.031, E3 -153105.566}
SPL {X  -159.990, Y  +384.326, Z    +0.000, E1  +359.760, E3 -153105.839}
SPL {X  -159.990, Y  +385.649, Z    +0.000, E1  +361.559, E3 -153105.851}
SPL {X  -159.990, Y  +388.306, Z    +0.000, E1  +365.901, E3 -153105.923}
SPL {X  -159.990, Y  +392.624, Z    +0.000, E1  +373.655, E3 -153106.172}
SPL {X  -159.990, Y  +398.511, Z    +0.000, E1  +384.979, E3 -153106.752}
SPL {X  -159.990, Y  +405.629, Z    +0.000, E1  +396.596, E3 -153107.883}
SPL {X  -159.990, Y  +417.919, Z    +0.000, E1  +410.108, E3 -153110.609}
SPL {X  -159.990, Y  +464.219, Z    +0.000, E1  +424.792, E3 -153128.668}
SPL {X  -159.990, Y  +601.948, Z    +0.000, E1  +428.261, E3 -153216.500}
SPL {X  -159.990, Y  +619.726, Z    +0.000, E1  +428.262, E3 -153231.561}
SPL {X  -159.990, Y  +636.530, Z    +0.000, E1  +428.257, E3 -153245.797}
SPL {X  -159.990, Y  +648.825, Z    +0.000, E1  +428.237, E3 -153256.256}
SPL {X  -159.990, Y  +661.441, Z    +0.000, E1  +428.256, E3 -153266.904}
SPL {X  -159.958, Y  +674.683, Z    +0.000, E1  +428.238, E3 -153278.166}
SPL {X  -159.269, Y  +686.675, Z    +0.000, E1  +428.163, E3 -153289.044}
SPL {X  -157.606, Y  +699.018, Z    +0.000, E1  +427.957, E3 -153301.228}
SPL {X  -155.210, Y  +710.317, Z    +0.000, E1  +427.656, E3 -153313.268}
SPL {X  -152.048, Y  +721.282, Z    +0.000, E1  +427.243, E3 -153325.760}
SPL {X  -148.485, Y  +731.073, Z    +0.000, E1  +426.748, E3 -153337.609}
SPL {X  -145.075, Y  +738.953, Z    +0.000, E1  +426.252, E3 -153347.601}
SPL {X  -141.751, Y  +745.686, Z    +0.000, E1  +425.756, E3 -153356.432}
SPL {X  -138.928, Y  +750.847, Z    +0.000, E1  +425.305, E3 -153363.401}
SPL {X  -136.328, Y  +755.234, Z    +0.000, E1  +424.898, E3 -153369.392}
SPL {X  -132.717, Y  +760.848, Z    +0.000, E1  +424.322, E3 -153377.165}
SPL {X  -128.512, Y  +766.796, Z    +0.000, E1  +423.597, E3 -153385.519}
SPL {X   -99.023, Y  +797.163, Z    +0.000, E1  +413.965, E3 -153487.349}
ENDSPLINE

SPLINE
SPL {X  -130.021, Y  +764.727, Z    +0.000, E1  +405.990, E3 -153626.868}
SPL {X  -148.409, Y  +731.264, Z    +0.000, E1  +396.685, E3 -153650.582}
SPL {X  -155.017, Y  +711.078, Z    +0.000, E1  +387.846, E3 -153657.643}
SPL {X  -158.217, Y  +695.254, Z    +0.000, E1  +378.896, E3 -153661.086}
SPL {X  -159.762, Y  +680.037, Z    +0.000, E1  +368.585, E3 -153662.802}
SPL {X  -159.990, Y  +671.255, Z    +0.000, E1  +361.602, E3 -153663.208}
SPL {X  -159.990, Y  +669.426, Z    +0.000, E1  +359.932, E3 -153663.228}
SPL {X  -159.990, Y  +666.879, Z    +0.000, E1  +356.292, E3 -153663.276}
SPL {X  -159.990, Y  +662.620, Z    +0.000, E1  +348.758, E3 -153663.477}
SPL {X  -159.990, Y  +657.714, Z    +0.000, E1  +339.502, E3 -153663.898}
SPL {X  -159.990, Y  +651.038, Z    +0.000, E1  +327.797, E3 -153664.800}
SPL {X  -159.990, Y  +637.243, Z    +0.000, E1  +311.500, E3 -153667.926}
SPL {X  -159.990, Y  +579.875, Z    +0.000, E1  +294.421, E3 -153690.784}
SPL {X  -159.990, Y  +453.091, Z    +0.000, E1  +291.862, E3 -153773.754}
SPL {X  -159.990, Y  +434.933, Z    +0.000, E1  +291.864, E3 -153789.248}
SPL {X  -159.990, Y  +420.071, Z    +0.000, E1  +291.886, E3 -153801.974}
SPL {X  -159.990, Y  +408.047, Z    +0.000, E1  +291.885, E3 -153812.221}
SPL {X  -159.990, Y  +395.904, Z    +0.000, E1  +291.881, E3 -153822.557}
SPL {X  -157.896, Y  +356.699, Z    +0.000, E1  +289.725, E3 -153834.866}
SPL {X  -156.475, Y  +349.148, Z    +0.000, E1  +290.612, E3 -153848.330}
SPL {X  -155.960, Y  +346.816, Z    +0.000, E1  +291.495, E3 -153857.492}
SPL {X  -154.913, Y  +342.515, Z    +0.000, E1  +292.501, E3 -153869.506}
SPL {X  -152.032, Y  +332.668, Z    +0.000, E1  +292.988, E3 -153881.497}
SPL {X  -148.460, Y  +322.864, Z    +0.000, E1  +293.452, E3 -153893.380}
SPL {X  -144.472, Y  +313.764, Z    +0.000, E1  +294.050, E3 -153905.043}
SPL {X  -140.755, Y  +306.442, Z    +0.000, E1  +294.606, E3 -153914.758}
SPL {X  -137.162, Y  +300.138, Z    +0.000, E1  +295.180, E3 -153923.366}
SPL {X  -134.303, Y  +295.555, Z    +0.000, E1  +295.659, E3 -153929.747}
SPL {X  -131.069, Y  +290.753, Z    +0.000, E1  +296.178, E3 -153936.481}
SPL {X  -127.815, Y  +286.271, Z    +0.000, E1  +296.784, E3 -153942.869}
SPL {X   -98.696, Y  +256.580, Z    +0.000, E1  +308.006, E3 -154078.420}
ENDSPLINE

SPLINE
SPL {X  -138.661, Y  +302.689, Z    +0.000, E1  +316.811, E3 -154196.148}
SPL {X  -154.202, Y  +339.857, Z    +0.000, E1  +330.366, E3 -154213.801}
SPL {X  -158.556, Y  +361.128, Z    +0.000, E1  +342.470, E3 -154218.323}
SPL {X  -159.663, Y  +372.278, Z    +0.000, E1  +350.186, E3 -154219.604}
SPL {X  -159.986, Y  +381.388, Z    +0.000, E1  +357.201, E3 -154220.076}
SPL {X  -159.990, Y  +384.492, Z    +0.000, E1  +359.986, E3 -154220.126}
SPL {X  -159.990, Y  +385.649, Z    +0.000, E1  +361.559, E3 -154220.137}
SPL {X  -159.990, Y  +389.563, Z    +0.000, E1  +367.931, E3 -154220.269}
SPL {X  -159.990, Y  +396.421, Z    +0.000, E1  +380.831, E3 -154220.814}
SPL {X  -159.990, Y  +405.629, Z    +0.000, E1  +396.596, E3 -154222.169}
SPL {X  -159.990, Y  +418.631, Z    +0.000, E1  +410.627, E3 -154225.116}
SPL {X  -159.990, Y  +468.459, Z    +0.000, E1  +425.348, E3 -154244.660}
SPL {X  -159.990, Y  +601.948, Z    +0.000, E1  +428.261, E3 -154330.786}
SPL {X  -159.990, Y  +619.726, Z    +0.000, E1  +428.262, E3 -154345.846}
SPL {X  -159.990, Y  +636.530, Z    +0.000, E1  +428.257, E3 -154360.083}
SPL {X  -159.990, Y  +648.825, Z    +0.000, E1  +428.237, E3 -154370.541}
SPL {X  -159.990, Y  +661.441, Z    +0.000, E1  +428.256, E3 -154381.190}
SPL {X  -159.958, Y  +674.683, Z    +0.000, E1  +428.238, E3 -154392.452}
SPL {X  -159.269, Y  +686.675, Z    +0.000, E1  +428.163, E3 -154403.330}
SPL {X  -158.119, Y  +695.895, Z    +0.000, E1  +428.003, E3 -154412.370}
SPL {X  -156.550, Y  +704.498, Z    +0.000, E1  +427.821, E3 -154421.261}
SPL {X  -154.561, Y  +712.826, Z    +0.000, E1  +427.549, E3 -154430.391}
SPL {X  -152.048, Y  +721.282, Z    +0.000, E1  +427.243, E3 -154440.046}
SPL {X  -148.485, Y  +731.073, Z    +0.000, E1  +426.748, E3 -154451.895}
SPL {X  -145.075, Y  +738.953, Z    +0.000, E1  +426.252, E3 -154461.887}
SPL {X  -141.751, Y  +745.686, Z    +0.000, E1  +425.756, E3 -154470.718}
SPL {X  -138.928, Y  +750.847, Z    +0.000, E1  +425.305, E3 -154477.687}
SPL {X  -136.328, Y  +755.234, Z    +0.000, E1  +424.898, E3 -154483.677}
SPL {X  -132.717, Y  +760.848, Z    +0.000, E1  +424.322, E3 -154491.450}
SPL {X  -128.512, Y  +766.796, Z    +0.000, E1  +423.597, E3 -154499.805}
SPL {X   -99.023, Y  +797.163, Z    +0.000, E1  +413.965, E3 -154601.635}
ENDSPLINE

SPLINE
SPL {X  -130.021, Y  +764.727, Z    +0.000, E1  +405.990, E3 -154741.154}
SPL {X  -148.409, Y  +731.264, Z    +0.000, E1  +396.685, E3 -154764.867}
SPL {X  -155.017, Y  +711.078, Z    +0.000, E1  +387.846, E3 -154771.928}
SPL {X  -158.217, Y  +695.254, Z    +0.000, E1  +378.896, E3 -154775.371}
SPL {X  -159.762, Y  +680.037, Z    +0.000, E1  +368.585, E3 -154777.088}
SPL {X  -159.990, Y  +671.255, Z    +0.000, E1  +361.602, E3 -154777.494}
SPL {X  -159.990, Y  +669.148, Z    +0.000, E1  +359.679, E3 -154777.516}
SPL {X  -159.990, Y  +666.130, Z    +0.000, E1  +354.946, E3 -154777.582}
SPL {X  -159.990, Y  +662.620, Z    +0.000, E1  +348.758, E3 -154777.762}
SPL {X  -159.990, Y  +657.714, Z    +0.000, E1  +339.502, E3 -154778.184}
SPL {X  -159.990, Y  +651.038, Z    +0.000, E1  +327.797, E3 -154779.086}
SPL {X  -159.990, Y  +637.243, Z    +0.000, E1  +311.500, E3 -154782.211}
SPL {X  -159.990, Y  +579.875, Z    +0.000, E1  +294.421, E3 -154805.070}
SPL {X  -159.990, Y  +453.091, Z    +0.000, E1  +291.862, E3 -154888.039}
SPL {X  -159.990, Y  +439.299, Z    +0.000, E1  +291.885, E3 -154899.852}
SPL {X  -159.990, Y  +424.060, Z    +0.000, E1  +291.860, E3 -154912.800}
SPL {X  -159.990, Y  +408.047, Z    +0.000, E1  +291.885, E3 -154926.507}
SPL {X  -159.990, Y  +395.904, Z    +0.000, E1  +291.881, E3 -154936.843}
SPL {X  -157.896, Y  +356.699, Z    +0.000, E1  +289.725, E3 -154949.152}
SPL {X  -156.475, Y  +349.148, Z    +0.000, E1  +290.612, E3 -154962.616}
SPL {X  -155.786, Y  +346.063, Z    +0.000, E1  +291.892, E3 -154975.911}
SPL {X  -154.401, Y  +340.583, Z    +0.000, E1  +292.675, E3 -154986.607}
SPL {X  -152.032, Y  +332.668, Z    +0.000, E1  +292.988, E3 -154995.783}
SPL {X  -149.782, Y  +326.266, Z    +0.000, E1  +293.308, E3 -155003.523}
SPL {X  -146.798, Y  +318.884, Z    +0.000, E1  +293.699, E3 -155012.703}
SPL {X  -143.755, Y  +312.276, Z    +0.000, E1  +294.175, E3 -155021.313}
SPL {X  -140.755, Y  +306.442, Z    +0.000, E1  +294.606, E3 -155029.044}
SPL {X  -137.162, Y  +300.138, Z    +0.000, E1  +295.180, E3 -155037.652}
SPL {X  -134.303, Y  +295.555, Z    +0.000, E1  +295.659, E3 -155044.033}
SPL {X  -132.067, Y  +292.194, Z    +0.000, E1  +296.034, E3 -155048.764}
SPL {X  -128.628, Y  +287.360, Z    +0.000, E1  +296.617, E3 -155055.587}
SPL {X   -98.696, Y  +256.580, Z    +0.000, E1  +308.006, E3 -155192.705}
ENDSPLINE

SPLINE
SPL {X  -138.661, Y  +302.689, Z    +0.000, E1  +316.811, E3 -155310.434}
SPL {X  -154.202, Y  +339.857, Z    +0.000, E1  +330.366, E3 -155328.087}
SPL {X  -158.556, Y  +361.128, Z    +0.000, E1  +342.470, E3 -155332.609}
SPL {X  -159.866, Y  +376.206, Z    +0.000, E1  +353.031, E3 -155334.138}
SPL {X  -159.990, Y  +384.326, Z    +0.000, E1  +359.760, E3 -155334.410}
SPL {X  -159.990, Y  +385.649, Z    +0.000, E1  +361.559, E3 -155334.423}
SPL {X  -159.990, Y  +389.563, Z    +0.000, E1  +367.931, E3 -155334.555}
SPL {X  -159.990, Y  +396.421, Z    +0.000, E1  +380.831, E3 -155335.100}
SPL {X  -159.990, Y  +405.629, Z    +0.000, E1  +396.596, E3 -155336.455}
SPL {X  -159.990, Y  +418.631, Z    +0.000, E1  +410.627, E3 -155339.402}
SPL {X  -159.990, Y  +468.459, Z    +0.000, E1  +425.348, E3 -155358.945}
SPL {X  -159.990, Y  +601.948, Z    +0.000, E1  +428.261, E3 -155445.071}
SPL {X  -159.990, Y  +619.726, Z    +0.000, E1  +428.262, E3 -155460.132}
SPL {X  -159.990, Y  +636.530, Z    +0.000, E1  +428.257, E3 -155474.368}
SPL {X  -159.990, Y  +653.116, Z    +0.000, E1  +428.255, E3 -155488.425}
SPL {X  -159.990, Y  +665.424, Z    +0.000, E1  +428.236, E3 -155498.889}
SPL {X  -159.958, Y  +674.683, Z    +0.000, E1  +428.238, E3 -155506.738}
SPL {X  -159.269, Y  +686.675, Z    +0.000, E1  +428.163, E3 -155517.615}
SPL {X  -158.119, Y  +695.895, Z    +0.000, E1  +428.003, E3 -155526.656}
SPL {X  -156.550, Y  +704.498, Z    +0.000, E1  +427.821, E3 -155535.546}
SPL {X  -154.561, Y  +712.826, Z    +0.000, E1  +427.549, E3 -155544.677}
SPL {X  -152.048, Y  +721.282, Z    +0.000, E1  +427.243, E3 -155554.332}
SPL {X  -148.485, Y  +731.073, Z    +0.000, E1  +426.748, E3 -155566.181}
SPL {X  -145.075, Y  +738.953, Z    +0.000, E1  +426.252, E3 -155576.172}
SPL {X  -141.751, Y  +745.686, Z    +0.000, E1  +425.756, E3 -155585.003}
SPL {X  -138.928, Y  +750.847, Z    +0.000, E1  +425.305, E3 -155591.973}
SPL {X  -135.390, Y  +756.743, Z    +0.000, E1  +424.775, E3 -155600.005}
SPL {X  -132.002, Y  +761.900, Z    +0.000, E1  +424.179, E3 -155607.236}
SPL {X  -128.512, Y  +766.796, Z    +0.000, E1  +423.597, E3 -155614.091}
SPL {X   -99.023, Y  +797.163, Z    +0.000, E1  +413.965, E3 -155715.920}
ENDSPLINE

SPLINE
SPL {X  -130.021, Y  +764.727, Z    +0.000, E1  +405.990, E3 -155855.440}
SPL {X  -148.409, Y  +731.264, Z    +0.000, E1  +396.685, E3 -155879.153}
SPL {X  -155.017, Y  +711.078, Z    +0.000, E1  +387.846, E3 -155886.214}
SPL {X  -158.217, Y  +695.254, Z    +0.000, E1  +378.896, E3 -155889.657}
SPL {X  -159.524, Y  +683.703, Z    +0.000, E1  +371.166, E3 -155891.099}
SPL {X  -159.986, Y  +672.621, Z    +0.000, E1  +362.847, E3 -155891.741}
SPL {X  -159.990, Y  +669.148, Z    +0.000, E1  +359.679, E3 -155891.802}
SPL {X  -159.990, Y  +666.130, Z    +0.000, E1  +354.946, E3 -155891.868}
SPL {X  -159.990, Y  +662.620, Z    +0.000, E1  +348.758, E3 -155892.048}
SPL {X  -159.990, Y  +657.714, Z    +0.000, E1  +339.502, E3 -155892.469}
SPL {X  -159.990, Y  +651.038, Z    +0.000, E1  +327.797, E3 -155893.372}
SPL {X  -159.990, Y  +642.324, Z    +0.000, E1  +316.129, E3 -155895.107}
SPL {X  -159.990, Y  +634.003, Z    +0.000, E1  +308.893, E3 -155897.382}
SPL {X  -159.990, Y  +579.875, Z    +0.000, E1  +294.421, E3 -155919.356}
SPL {X  -159.990, Y  +453.091, Z    +0.000, E1  +291.862, E3 -156002.325}
SPL {X  -159.990, Y  +434.933, Z    +0.000, E1  +291.864, E3 -156017.819}
SPL {X  -159.990, Y  +420.071, Z    +0.000, E1  +291.886, E3 -156030.545}
SPL {X  -159.990, Y  +408.047, Z    +0.000, E1  +291.885, E3 -156040.792}
SPL {X  -159.990, Y  +395.904, Z    +0.000, E1  +291.881, E3 -156051.128}
SPL {X  -157.896, Y  +356.699, Z    +0.000, E1  +289.725, E3 -156063.438}
SPL {X  -156.475, Y  +349.148, Z    +0.000, E1  +290.612, E3 -156076.902}
SPL {X  -155.786, Y  +346.063, Z    +0.000, E1  +291.892, E3 -156090.196}
SPL {X  -154.401, Y  +340.583, Z    +0.000, E1  +292.675, E3 -156100.893}
SPL {X  -152.032, Y  +332.668, Z    +0.000, E1  +292.988, E3 -156110.069}
SPL {X  -148.460, Y  +322.864, Z    +0.000, E1  +293.452, E3 -156121.951}
SPL {X  -144.472, Y  +313.764, Z    +0.000, E1  +294.050, E3 -156133.615}
SPL {X  -140.755, Y  +306.442, Z    +0.000, E1  +294.606, E3 -156143.329}
SPL {X  -137.162, Y  +300.138, Z    +0.000, E1  +295.180, E3 -156151.937}
SPL {X  -134.303, Y  +295.555, Z    +0.000, E1  +295.659, E3 -156158.318}
SPL {X  -131.069, Y  +290.753, Z    +0.000, E1  +296.178, E3 -156165.052}
SPL {X  -127.815, Y  +286.271, Z    +0.000, E1  +296.784, E3 -156171.440}
SPL {X   -99.903, Y  +257.535, Z    +0.000, E1  +308.539, E3 -156318.736}
ENDSPLINE

SPLINE
SPL {X  -141.433, Y  +307.709, Z    +0.000, E1  +318.157, E3 -156428.533}
SPL {X  -154.202, Y  +339.857, Z    +0.000, E1  +330.366, E3 -156442.373}
SPL {X  -158.556, Y  +361.128, Z    +0.000, E1  +342.470, E3 -156446.894}
SPL {X  -159.663, Y  +372.278, Z    +0.000, E1  +350.186, E3 -156448.176}
SPL {X  -159.986, Y  +381.388, Z    +0.000, E1  +357.201, E3 -156448.647}
SPL {X  -159.990, Y  +384.932, Z    +0.000, E1  +360.381, E3 -156448.702}
SPL {X  -159.990, Y  +389.563, Z    +0.000, E1  +367.931, E3 -156448.841}
SPL {X  -159.990, Y  +396.421, Z    +0.000, E1  +380.831, E3 -156449.386}
SPL {X  -159.990, Y  +405.629, Z    +0.000, E1  +396.596, E3 -156450.740}
SPL {X  -159.990, Y  +417.919, Z    +0.000, E1  +410.108, E3 -156453.466}
SPL {X  -159.990, Y  +464.219, Z    +0.000, E1  +424.792, E3 -156471.525}
SPL {X  -159.990, Y  +601.948, Z    +0.000, E1  +428.261, E3 -156559.357}
SPL {X  -159.990, Y  +614.867, Z    +0.000, E1  +428.239, E3 -156570.356}
SPL {X  -159.990, Y  +627.954, Z    +0.000, E1  +428.256, E3 -156581.400}
SPL {X  -159.990, Y  +640.176, Z    +0.000, E1  +428.239, E3 -156591.779}
SPL {X  -159.990, Y  +653.116, Z    +0.000, E1  +428.255, E3 -156602.710}
SPL {X  -159.990, Y  +665.424, Z    +0.000, E1  +428.236, E3 -156613.175}
SPL {X  -159.958, Y  +674.683, Z    +0.000, E1  +428.238, E3 -156621.024}
SPL {X  -159.269, Y  +686.675, Z    +0.000, E1  +428.163, E3 -156631.901}
SPL {X  -158.119, Y  +695.895, Z    +0.000, E1  +428.003, E3 -156640.942}
SPL {X  -156.550, Y  +704.498, Z    +0.000, E1  +427.821, E3 -156649.832}
SPL {X  -154.561, Y  +712.826, Z    +0.000, E1  +427.549, E3 -156658.963}
SPL {X  -152.048, Y  +721.282, Z    +0.000, E1  +427.243, E3 -156668.617}
SPL {X  -148.485, Y  +731.073, Z    +0.000, E1  +426.748, E3 -156680.466}
SPL {X  -145.075, Y  +738.953, Z    +0.000, E1  +426.252, E3 -156690.458}
SPL {X  -141.751, Y  +745.686, Z    +0.000, E1  +425.756, E3 -156699.289}
SPL {X  -138.928, Y  +750.847, Z    +0.000, E1  +425.305, E3 -156706.258}
SPL {X  -136.328, Y  +755.234, Z    +0.000, E1  +424.898, E3 -156712.249}
SPL {X  -132.717, Y  +760.848, Z    +0.000, E1  +424.322, E3 -156720.022}
SPL {X  -129.778, Y  +765.065, Z    +0.000, E1  +423.787, E3 -156725.977}
SPL {X  -127.600, Y  +768.014, Z    +0.000, E1  +423.408, E3 -156730.123}
SPL {X   -99.023, Y  +797.163, Z    +0.000, E1  +413.965, E3 -156830.206}
ENDSPLINE

SPLINE
SPL {X  -130.021, Y  +764.727, Z    +0.000, E1  +405.990, E3 -156969.725}
SPL {X  -148.409, Y  +731.264, Z    +0.000, E1  +396.685, E3 -156993.439}
SPL {X  -155.017, Y  +711.078, Z    +0.000, E1  +387.846, E3 -157000.500}
SPL {X  -158.217, Y  +695.254, Z    +0.000, E1  +378.896, E3 -157003.943}
SPL {X  -159.762, Y  +680.037, Z    +0.000, E1  +368.585, E3 -157005.660}
SPL {X  -159.990, Y  +671.255, Z    +0.000, E1  +361.602, E3 -157006.065}
SPL {X  -159.990, Y  +669.148, Z    +0.000, E1  +359.679, E3 -157006.088}
SPL {X  -159.990, Y  +666.130, Z    +0.000, E1  +354.946, E3 -157006.154}
SPL {X  -159.990, Y  +662.620, Z    +0.000, E1  +348.758, E3 -157006.334}
SPL {X  -159.990, Y  +657.714, Z    +0.000, E1  +339.502, E3 -157006.755}
SPL {X  -159.990, Y  +651.038, Z    +0.000, E1  +327.797, E3 -157007.658}
SPL {X  -159.990, Y  +637.243, Z    +0.000, E1  +311.500, E3 -157010.783}
SPL {X  -159.990, Y  +579.875, Z    +0.000, E1  +294.421, E3 -157033.641}
SPL {X  -159.990, Y  +453.091, Z    +0.000, E1  +291.862, E3 -157116.611}
SPL {X  -159.990, Y  +434.933, Z    +0.000, E1  +291.864, E3 -157132.105}
SPL {X  -159.990, Y  +420.071, Z    +0.000, E1  +291.886, E3 -157144.831}
SPL {X  -159.990, Y  +408.047, Z    +0.000, E1  +291.885, E3 -157155.078}
SPL {X  -159.990, Y  +395.904, Z    +0.000, E1  +291.881, E3 -157165.414}
SPL {X  -157.896, Y  +356.699, Z    +0.000, E1  +289.725, E3 -157177.724}
SPL {X  -156.475, Y  +349.148, Z    +0.000, E1  +290.612, E3 -157191.188}
SPL {X  -155.786, Y  +346.063, Z    +0.000, E1  +291.892, E3 -157204.482}
SPL {X  -153.671, Y  +337.981, Z    +0.000, E1  +292.746, E3 -157218.102}
SPL {X  -150.407, Y  +327.960, Z    +0.000, E1  +293.203, E3 -157229.991}
SPL {X  -146.798, Y  +318.884, Z    +0.000, E1  +293.699, E3 -157241.275}
SPL {X  -142.741, Y  +310.238, Z    +0.000, E1  +294.301, E3 -157252.534}
SPL {X  -139.838, Y  +304.768, Z    +0.000, E1  +294.773, E3 -157259.917}
SPL {X  -137.162, Y  +300.138, Z    +0.000, E1  +295.180, E3 -157266.223}
SPL {X  -132.996, Y  +293.568, Z    +0.000, E1  +295.842, E3 -157275.357}
SPL {X  -128.628, Y  +287.360, Z    +0.000, E1  +296.617, E3 -157284.159}
SPL {X   -98.696, Y  +256.580, Z    +0.000, E1  +308.006, E3 -157421.277}
ENDSPLINE

SPLINE
SPL {X  -138.661, Y  +302.689, Z    +0.000, E1  +316.811, E3 -157539.005}
SPL {X  -154.202, Y  +339.857, Z    +0.000, E1  +330.366, E3 -157556.658}
SPL {X  -158.556, Y  +361.128, Z    +0.000, E1  +342.470, E3 -157561.180}
SPL {X  -159.866, Y  +376.206, Z    +0.000, E1  +353.031, E3 -157562.709}
SPL {X  -159.990, Y  +384.789, Z    +0.000, E1  +360.146, E3 -157562.986}
SPL {X  -159.990, Y  +388.306, Z    +0.000, E1  +365.901, E3 -157563.066}
SPL {X  -159.990, Y  +392.624, Z    +0.000, E1  +373.655, E3 -157563.315}
SPL {X  -159.990, Y  +398.511, Z    +0.000, E1  +384.979, E3 -157563.895}
SPL {X  -159.990, Y  +405.629, Z    +0.000, E1  +396.596, E3 -157565.026}
SPL {X  -159.990, Y  +418.631, Z    +0.000, E1  +410.627, E3 -157567.973}
SPL {X  -159.990, Y  +468.459, Z    +0.000, E1  +425.348, E3 -157587.517}
SPL {X  -159.990, Y  +601.948, Z    +0.000, E1  +428.261, E3 -157673.643}
SPL {X  -159.990, Y  +619.726, Z    +0.000, E1  +428.262, E3 -157688.704}
SPL {X  -159.990, Y  +636.530, Z    +0.000, E1  +428.257, E3 -157702.940}
SPL {X  -159.990, Y  +648.825, Z    +0.000, E1  +428.237, E3 -157713.398}
SPL {X  -159.990, Y  +661.441, Z    +0.000, E1  +428.256, E3 -157724.047}
SPL {X  -159.958, Y  +674.683, Z    +0.000, E1  +428.238, E3 -157735.309}
SPL {X  -159.269, Y  +686.675, Z    +0.000, E1  +428.163, E3 -157746.187}
SPL {X  -157.606, Y  +699.018, Z    +0.000, E1  +427.957, E3 -157758.370}
SPL {X  -155.210, Y  +710.317, Z    +0.000, E1  +427.656, E3 -157770.410}
SPL {X  -152.048, Y  +721.282, Z    +0.000, E1  +427.243, E3 -157782.903}
SPL {X  -148.485, Y  +731.073, Z    +0.000, E1  +426.748, E3 -157794.752}
SPL {X  -145.075, Y  +738.953, Z    +0.000, E1  +426.252, E3 -157804.744}
SPL {X  -141.751, Y  +745.686, Z    +0.000, E1  +425.756, E3 -157813.575}
SPL {X  -138.928, Y  +750.847, Z    +0.000, E1  +425.305, E3 -157820.544}
SPL {X  -136.328, Y  +755.234, Z    +0.000, E1  +424.898, E3 -157826.534}
SPL {X  -132.717, Y  +760.848, Z    +0.000, E1  +424.322, E3 -157834.308}
SPL {X  -128.512, Y  +766.796, Z    +0.000, E1  +423.597, E3 -157842.662}
SPL {X   -99.023, Y  +797.163, Z    +0.000, E1  +413.965, E3 -157944.492}
ENDSPLINE

SPLINE
SPL {X  -130.021, Y  +764.727, Z    +0.000, E1  +405.990, E3 -158084.011}
SPL {X  -148.409, Y  +731.264, Z    +0.000, E1  +396.685, E3 -158107.725}
SPL {X  -155.017, Y  +711.078, Z    +0.000, E1  +387.846, E3 -158114.786}
SPL {X  -158.217, Y  +695.254, Z    +0.000, E1  +378.896, E3 -158118.228}
SPL {X  -159.762, Y  +680.037, Z    +0.000, E1  +368.585, E3 -158119.945}
SPL {X  -159.990, Y  +671.255, Z    +0.000, E1  +361.602, E3 -158120.351}
SPL {X  -159.990, Y  +669.426, Z    +0.000, E1  +359.932, E3 -158120.371}
SPL {X  -159.990, Y  +666.879, Z    +0.000, E1  +356.292, E3 -158120.418}
SPL {X  -159.990, Y  +662.620, Z    +0.000, E1  +348.758, E3 -158120.620}
SPL {X  -159.990, Y  +657.714, Z    +0.000, E1  +339.502, E3 -158121.041}
SPL {X  -159.990, Y  +651.038, Z    +0.000, E1  +327.797, E3 -158121.943}
SPL {X  -159.990, Y  +637.243, Z    +0.000, E1  +311.500, E3 -158125.068}
SPL {X  -159.990, Y  +579.875, Z    +0.000, E1  +294.421, E3 -158147.927}
SPL {X  -159.990, Y  +453.091, Z    +0.000, E1  +291.862, E3 -158230.897}
SPL {X  -159.990, Y  +434.933, Z    +0.000, E1  +291.864, E3 -158246.390}
SPL {X  -159.990, Y  +420.071, Z    +0.000, E1  +291.886, E3 -158259.116}
SPL {X  -159.990, Y  +408.047, Z    +0.000, E1  +291.885, E3 -158269.364}
SPL {X  -159.990, Y  +395.904, Z    +0.000, E1  +291.881, E3 -158279.700}
SPL {X  -157.896, Y  +356.699, Z    +0.000, E1  +289.725, E3 -158292.009}
SPL {X  -156.475, Y  +349.148, Z    +0.000, E1  +290.612, E3 -158305.473}
SPL {X  -155.960, Y  +346.816, Z    +0.000, E1  +291.495, E3 -158314.635}
SPL {X  -154.913, Y  +342.515, Z    +0.000, E1  +292.501, E3 -158326.649}
SPL {X  -152.032, Y  +332.668, Z    +0.000, E1  +292.988, E3 -158338.640}
SPL {X  -148.460, Y  +322.864, Z    +0.000, E1  +293.452, E3 -158350.523}
SPL {X  -144.472, Y  +313.764, Z    +0.000, E1  +294.050, E3 -158362.186}
SPL {X  -140.755, Y  +306.442, Z    +0.000, E1  +294.606, E3 -158371.901}
SPL {X  -137.162, Y  +300.138, Z    +0.000, E1  +295.180, E3 -158380.509}
SPL {X  -134.303, Y  +295.555, Z    +0.000, E1  +295.659, E3 -158386.890}
SPL {X  -131.069, Y  +290.753, Z    +0.000, E1  +296.178, E3 -158393.623}
SPL {X  -127.815, Y  +286.271, Z    +0.000, E1  +296.784, E3 -158400.012}
SPL {X   -98.696, Y  +256.580, Z    +0.000, E1  +308.006, E3 -158535.562}
ENDSPLINE

SPLINE
SPL {X  -138.661, Y  +302.689, Z    +0.000, E1  +316.811, E3 -158653.291}
SPL {X  -154.202, Y  +339.857, Z    +0.000, E1  +330.366, E3 -158670.944}
SPL {X  -158.556, Y  +361.128, Z    +0.000, E1  +342.470, E3 -158675.466}
SPL {X  -159.663, Y  +372.278, Z    +0.000, E1  +350.186, E3 -158676.747}
SPL {X  -159.986, Y  +381.388, Z    +0.000, E1  +357.201, E3 -158677.218}
SPL {X  -159.990, Y  +384.492, Z    +0.000, E1  +359.986, E3 -158677.269}
SPL {X  -159.990, Y  +385.649, Z    +0.000, E1  +361.559, E3 -158677.280}
SPL {X  -159.990, Y  +389.563, Z    +0.000, E1  +367.931, E3 -158677.412}
SPL {X  -159.990, Y  +396.421, Z    +0.000, E1  +380.831, E3 -158677.957}
SPL {X  -159.990, Y  +405.629, Z    +0.000, E1  +396.596, E3 -158679.312}
SPL {X  -159.990, Y  +418.631, Z    +0.000, E1  +410.627, E3 -158682.259}
SPL {X  -159.990, Y  +468.459, Z    +0.000, E1  +425.348, E3 -158701.803}
SPL {X  -159.990, Y  +601.948, Z    +0.000, E1  +428.261, E3 -158787.929}
SPL {X  -159.990, Y  +619.726, Z    +0.000, E1  +428.262, E3 -158802.989}
SPL {X  -159.990, Y  +636.530, Z    +0.000, E1  +428.257, E3 -158817.225}
SPL {X  -159.990, Y  +648.825, Z    +0.000, E1  +428.237, E3 -158827.684}
SPL {X  -159.990, Y  +661.441, Z    +0.000, E1  +428.256, E3 -158838.332}
SPL {X  -159.958, Y  +674.683, Z    +0.000, E1  +428.238, E3 -158849.595}
SPL {X  -159.269, Y  +686.675, Z    +0.000, E1  +428.163, E3 -158860.472}
SPL {X  -158.119, Y  +695.895, Z    +0.000, E1  +428.003, E3 -158869.513}
SPL {X  -156.550, Y  +704.498, Z    +0.000, E1  +427.821, E3 -158878.403}
SPL {X  -153.468, Y  +716.715, Z    +0.000, E1  +427.444, E3 -158891.866}
SPL {X  -149.840, Y  +727.578, Z    +0.000, E1  +426.935, E3 -158904.742}
SPL {X  -145.768, Y  +737.444, Z    +0.000, E1  +426.379, E3 -158917.044}
SPL {X  -141.751, Y  +745.686, Z    +0.000, E1  +425.756, E3 -158927.860}
SPL {X  -138.928, Y  +750.847, Z    +0.000, E1  +425.305, E3 -158934.830}
SPL {X  -136.328, Y  +755.234, Z    +0.000, E1  +424.898, E3 -158940.820}
SPL {X  -132.717, Y  +760.848, Z    +0.000, E1  +424.322, E3 -158948.593}
SPL {X  -128.512, Y  +766.796, Z    +0.000, E1  +423.597, E3 -158956.948}
SPL {X   -99.023, Y  +797.163, Z    +0.000, E1  +413.965, E3 -159058.777}
ENDSPLINE

SPLINE
SPL {X  -130.021, Y  +764.727, Z    +0.000, E1  +405.990, E3 -159198.297}
SPL {X  -148.409, Y  +731.264, Z    +0.000, E1  +396.685, E3 -159222.010}
SPL {X  -155.017, Y  +711.078, Z    +0.000, E1  +387.846, E3 -159229.071}
SPL {X  -158.217, Y  +695.254, Z    +0.000, E1  +378.896, E3 -159232.514}
SPL {X  -159.762, Y  +680.037, Z    +0.000, E1  +368.585, E3 -159234.231}
SPL {X  -159.990, Y  +671.255, Z    +0.000, E1  +361.602, E3 -159234.637}
SPL {X  -159.990, Y  +669.426, Z    +0.000, E1  +359.932, E3 -159234.656}
SPL {X  -159.990, Y  +666.879, Z    +0.000, E1  +356.292, E3 -159234.704}
SPL {X  -159.990, Y  +662.620, Z    +0.000, E1  +348.758, E3 -159234.905}
SPL {X  -159.990, Y  +657.714, Z    +0.000, E1  +339.502, E3 -159235.327}
SPL {X  -159.990, Y  +651.038, Z    +0.000, E1  +327.797, E3 -159236.229}
SPL {X  -159.990, Y  +637.243, Z    +0.000, E1  +311.500, E3 -159239.354}
SPL {X  -159.990, Y  +579.875, Z    +0.000, E1  +294.421, E3 -159262.213}
SPL {X  -159.990, Y  +453.091, Z    +0.000, E1  +291.862, E3 -159345.182}
SPL {X  -159.990, Y  +434.933, Z    +0.000, E1  +291.864, E3 -159360.676}
SPL {X  -159.990, Y  +420.071, Z    +0.000, E1  +291.886, E3 -159373.402}
SPL {X  -159.990, Y  +408.047, Z    +0.000, E1  +291.885, E3 -159383.650}
SPL {X  -159.990, Y  +395.904, Z    +0.000, E1  +291.881, E3 -159393.986}
SPL {X  -157.896, Y  +356.699, Z    +0.000, E1  +289.725, E3 -159406.295}
SPL {X  -156.475, Y  +349.148, Z    +0.000, E1  +290.612, E3 -159419.759}
SPL {X  -155.786, Y  +346.063, Z    +0.000, E1  +291.892, E3 -159433.053}
SPL {X  -153.671, Y  +337.981, Z    +0.000, E1  +292.746, E3 -159446.673}
SPL {X  -150.407, Y  +327.960, Z    +0.000, E1  +293.203, E3 -159458.562}
SPL {X  -147.566, Y  +320.686, Z    +0.000, E1  +293.613, E3 -159467.602}
SPL {X  -144.472, Y  +313.764, Z    +0.000, E1  +294.050, E3 -159476.472}
SPL {X  -140.755, Y  +306.442, Z    +0.000, E1  +294.606, E3 -159486.186}
SPL {X  -137.162, Y  +300.138, Z    +0.000, E1  +295.180, E3 -159494.795}
SPL {X  -132.996, Y  +293.568, Z    +0.000, E1  +295.842, E3 -159503.929}
SPL {X  -128.628, Y  +287.360, Z    +0.000, E1  +296.617, E3 -159512.730}
SPL {X   -98.696, Y  +256.580, Z    +0.000, E1  +308.006, E3 -159649.848}
ENDSPLINE

